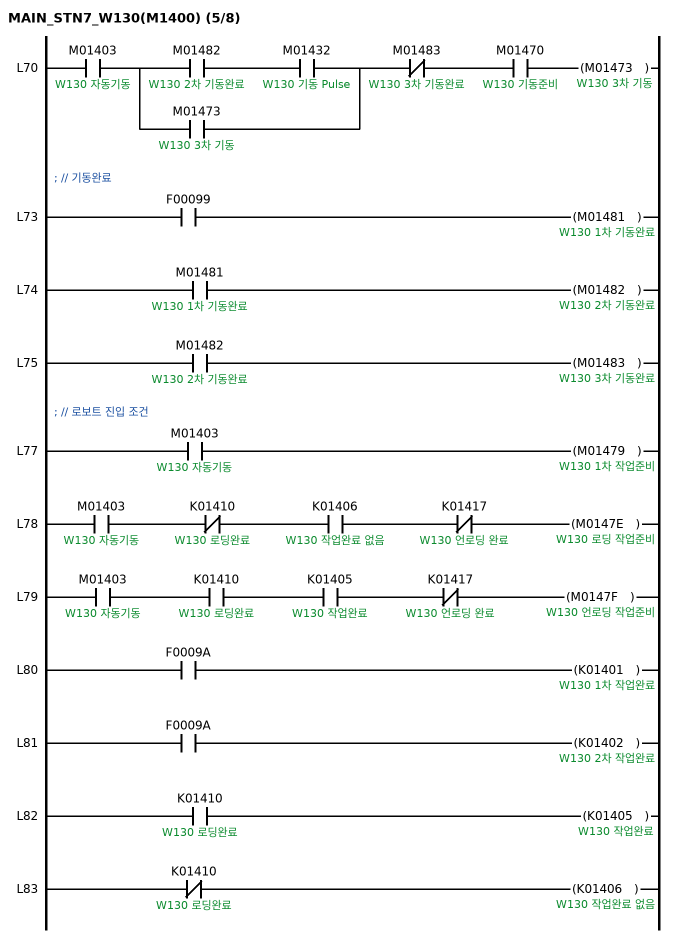
[picture p144: MAIN_STN7_W130(M1400) rungs L70-L83]
; L70
LOAD      M01403	// W130 자동기동
LOAD      M01482	// W130 2차 기동완료
AND       M01432	// W130 기동 Pulse
OR        M01473	// W130 3차 기동
AND LOAD
AND NOT   M01483	// W130 3차 기동완료
AND       M01470	// W130 기동준비
OUT       M01473	// W130 3차 기동
//   // 기동완료
; L73
LOAD      F00099
OUT       M01481	// W130 1차 기동완료
; L74
LOAD      M01481	// W130 1차 기동완료
OUT       M01482	// W130 2차 기동완료
; L75
LOAD      M01482	// W130 2차 기동완료
OUT       M01483	// W130 3차 기동완료
//   // 로보트 진입 조건
; L77
LOAD      M01403	// W130 자동기동
OUT       M01479	// W130 1차 작업준비
; L78
LOAD      M01403	// W130 자동기동
AND NOT   K01410	// W130 로딩완료
AND       K01406	// W130 작업완료 없음
AND NOT   K01417	// W130 언로딩 완료
OUT       M0147E	// W130 로딩 작업준비
; L79
LOAD      M01403	// W130 자동기동
AND       K01410	// W130 로딩완료
AND       K01405	// W130 작업완료
AND NOT   K01417	// W130 언로딩 완료
OUT       M0147F	// W130 언로딩 작업준비
; L80
LOAD      F0009A
OUT       K01401	// W130 1차 작업완료
; L81
LOAD      F0009A
OUT       K01402	// W130 2차 작업완료
; L82
LOAD      K01410	// W130 로딩완료
OUT       K01405	// W130 작업완료
; L83
LOAD NOT  K01410	// W130 로딩완료
OUT       K01406	// W130 작업완료 없음

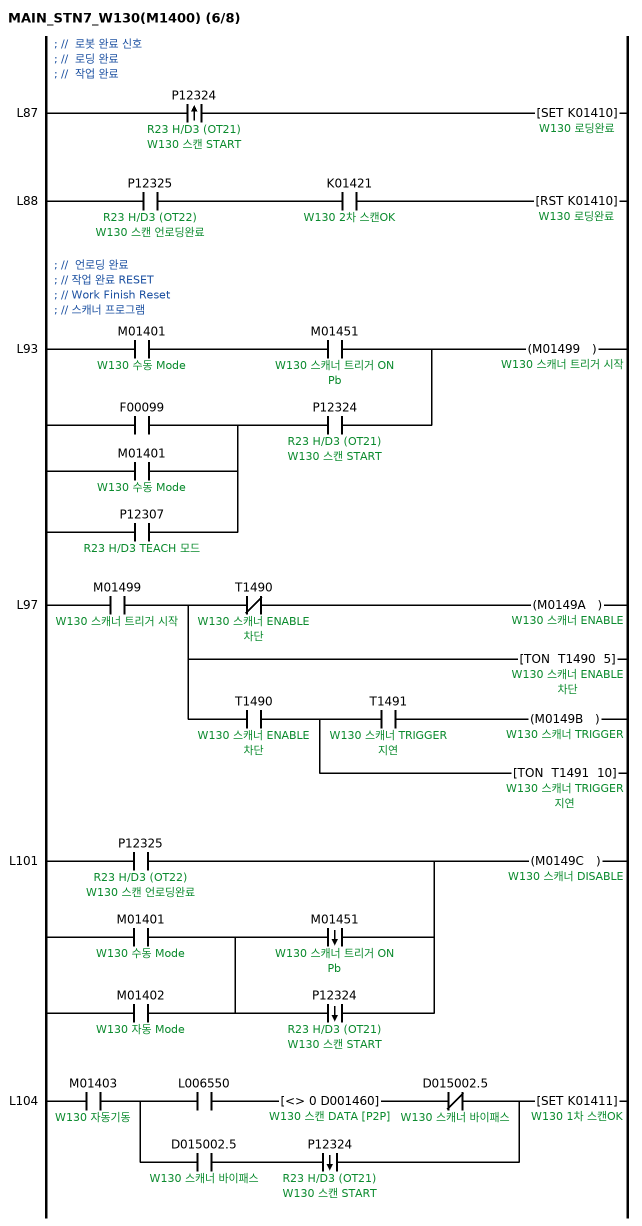
//   //  로봇 완료 신호
//   //  로딩 완료
//   //  작업 완료
; L87
LOADP     P12324	// R23 H/D3 (OT21) W130 스캔 START
SET       K01410	// W130 로딩완료
; L88
LOAD      P12325	// R23 H/D3 (OT22) W130 스캔 언로딩완료
AND       K01421	// W130 2차 스캔OK
RST       K01410	// W130 로딩완료
//   //  언로딩 완료
//     // 작업 완료 RESET
//   // Work Finish Reset
//   // 스캐너 프로그램
; L93
LOAD      M01401	// W130 수동 Mode
AND       M01451	// W130 스캐너 트리거 ON Pb
LOAD      F00099
OR        M01401	// W130 수동 Mode
OR        P12307	// R23 H/D3 TEACH 모드
AND       P12324	// R23 H/D3 (OT21) W130 스캔 START
OR LOAD
OUT       M01499	// W130 스캐너 트리거 시작
; L97
LOAD      M01499	// W130 스캐너 트리거 시작
MPUSH
AND NOT   T1490	// W130 스캐너 ENABLE 차단
OUT       M0149A	// W130 스캐너 ENABLE
MPOP
TON       T1490 5	// W130 스캐너 ENABLE 차단
AND       T1490	// W130 스캐너 ENABLE 차단
MPUSH
AND       T1491	// W130 스캐너 TRIGGER 지연
OUT       M0149B	// W130 스캐너 TRIGGER
MPOP
TON       T1491 10	// W130 스캐너 TRIGGER 지연
; L101
LOAD      P12325	// R23 H/D3 (OT22) W130 스캔 언로딩완료
LOAD      M01401	// W130 수동 Mode
OR        M01402	// W130 자동 Mode
LOADN     M01451	// W130 스캐너 트리거 ON Pb
ORN       P12324	// R23 H/D3 (OT21) W130 스캔 START
AND LOAD
OR LOAD
OUT       M0149C	// W130 스캐너 DISABLE
; L104
LOAD      M01403	// W130 자동기동
LOAD      L006550
AND<>     0 D001460	// W130 스캔 DATA [P2P]
AND NOT   D015002.5	// W130 스캐너 바이패스
LOAD      D015002.5	// W130 스캐너 바이패스
ANDN      P12324	// R23 H/D3 (OT21) W130 스캔 START
OR LOAD
AND LOAD
SET       K01411	// W130 1차 스캔OK

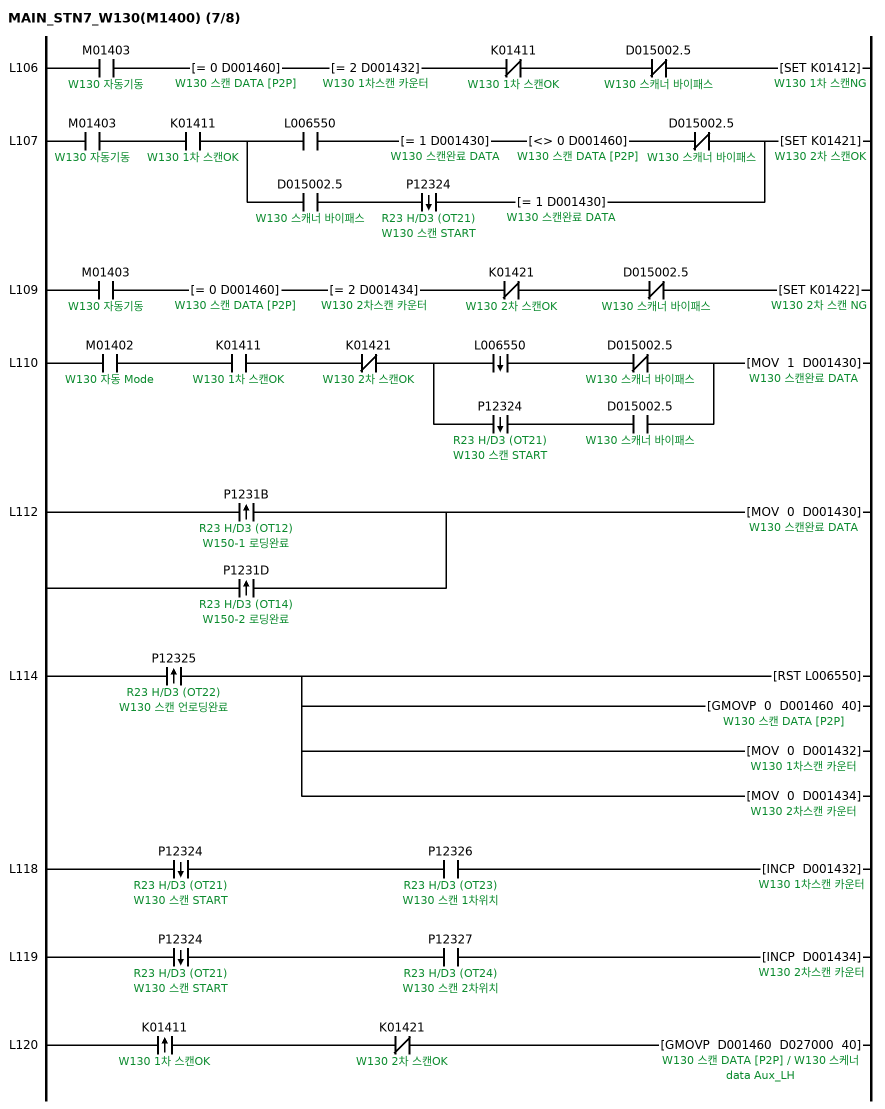
; L106
LOAD      M01403	// W130 자동기동
AND=      0 D001460	// W130 스캔 DATA [P2P]
AND=      2 D001432	// W130 1차스캔 카운터
AND NOT   K01411	// W130 1차 스캔OK
AND NOT   D015002.5	// W130 스캐너 바이패스
SET       K01412	// W130 1차 스캔NG
; L107
LOAD      M01403	// W130 자동기동
AND       K01411	// W130 1차 스캔OK
LOAD      L006550
AND=      1 D001430	// W130 스캔완료 DATA
AND<>     0 D001460	// W130 스캔 DATA [P2P]
AND NOT   D015002.5	// W130 스캐너 바이패스
LOAD      D015002.5	// W130 스캐너 바이패스
ANDN      P12324	// R23 H/D3 (OT21) W130 스캔 START
AND=      1 D001430	// W130 스캔완료 DATA
OR LOAD
AND LOAD
SET       K01421	// W130 2차 스캔OK
; L109
LOAD      M01403	// W130 자동기동
AND=      0 D001460	// W130 스캔 DATA [P2P]
AND=      2 D001434	// W130 2차스캔 카운터
AND NOT   K01421	// W130 2차 스캔OK
AND NOT   D015002.5	// W130 스캐너 바이패스
SET       K01422	// W130 2차 스캔 NG
; L110
LOAD      M01402	// W130 자동 Mode
AND       K01411	// W130 1차 스캔OK
AND NOT   K01421	// W130 2차 스캔OK
LOADN     L006550
AND NOT   D015002.5	// W130 스캐너 바이패스
LOADN     P12324	// R23 H/D3 (OT21) W130 스캔 START
AND       D015002.5	// W130 스캐너 바이패스
OR LOAD
AND LOAD
MOV       1 D001430	// W130 스캔완료 DATA
; L112
LOADP     P1231B	// R23 H/D3 (OT12) W150-1 로딩완료
ORP       P1231D	// R23 H/D3 (OT14) W150-2 로딩완료
MOV       0 D001430	// W130 스캔완료 DATA
; L114
LOADP     P12325	// R23 H/D3 (OT22) W130 스캔 언로딩완료
RST       L006550
GMOVP     0 D001460 40	// W130 스캔 DATA [P2P]
MOV       0 D001432	// W130 1차스캔 카운터
MOV       0 D001434	// W130 2차스캔 카운터
; L118
LOADN     P12324	// R23 H/D3 (OT21) W130 스캔 START
AND       P12326	// R23 H/D3 (OT23) W130 스캔 1차위치
INCP      D001432	// W130 1차스캔 카운터
; L119
LOADN     P12324	// R23 H/D3 (OT21) W130 스캔 START
AND       P12327	// R23 H/D3 (OT24) W130 스캔 2차위치
INCP      D001434	// W130 2차스캔 카운터
; L120
LOADP     K01411	// W130 1차 스캔OK
AND NOT   K01421	// W130 2차 스캔OK
GMOVP     D001460 D027000 40	// W130 스캔 DATA [P2P] / W130 스케너 data Aux_LH

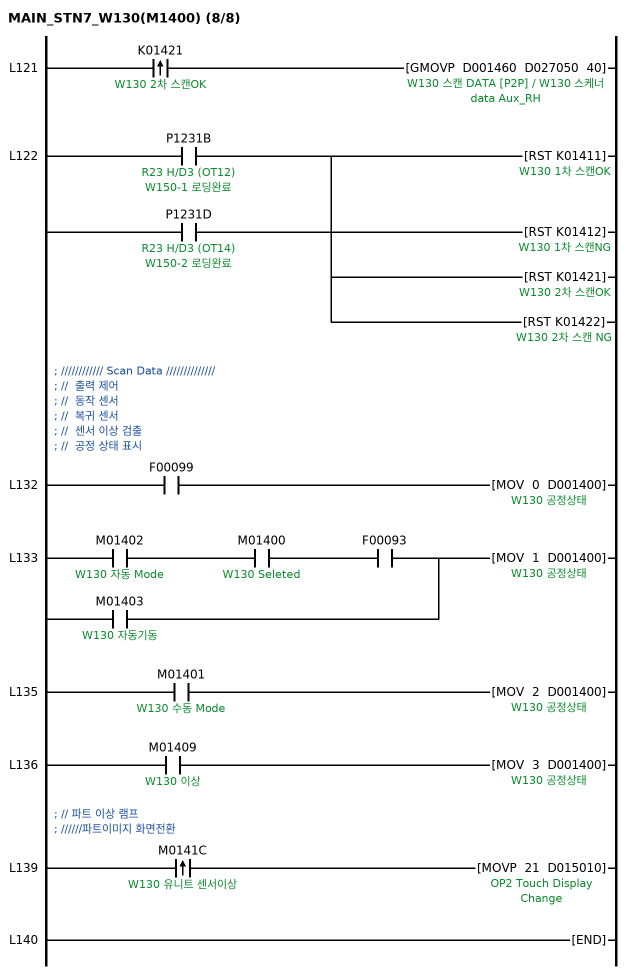
; L121
LOADP     K01421	// W130 2차 스캔OK
GMOVP     D001460 D027050 40	// W130 스캔 DATA [P2P] / W130 스케너 data Aux_RH
; L122
LOAD      P1231B	// R23 H/D3 (OT12) W150-1 로딩완료
OR        P1231D	// R23 H/D3 (OT14) W150-2 로딩완료
RST       K01411	// W130 1차 스캔OK
RST       K01412	// W130 1차 스캔NG
RST       K01421	// W130 2차 스캔OK
RST       K01422	// W130 2차 스캔 NG
// //////////// Scan Data //////////////
//     //  출력 제어
//   //  동작 센서
//   //  복귀 센서
//     //  센서 이상 검출
//   //  공정 상태 표시
; L132
LOAD      F00099
MOV       0 D001400	// W130 공정상태
; L133
LOAD      M01402	// W130 자동 Mode
AND       M01400	// W130 Seleted
AND       F00093
OR        M01403	// W130 자동기동
MOV       1 D001400	// W130 공정상태
; L135
LOAD      M01401	// W130 수동 Mode
MOV       2 D001400	// W130 공정상태
; L136
LOAD      M01409	// W130 이상
MOV       3 D001400	// W130 공정상태
//   // 파트 이상 램프
// //////파트이미지 화면전환
; L139
LOADP     M0141C	// W130 유니트 센서이상
MOVP      21 D015010	// OP2 Touch Display Change
; L140
END

PROGRAM MAIN_STN8_W150-1(M800) (task: 스캔 프로그램)

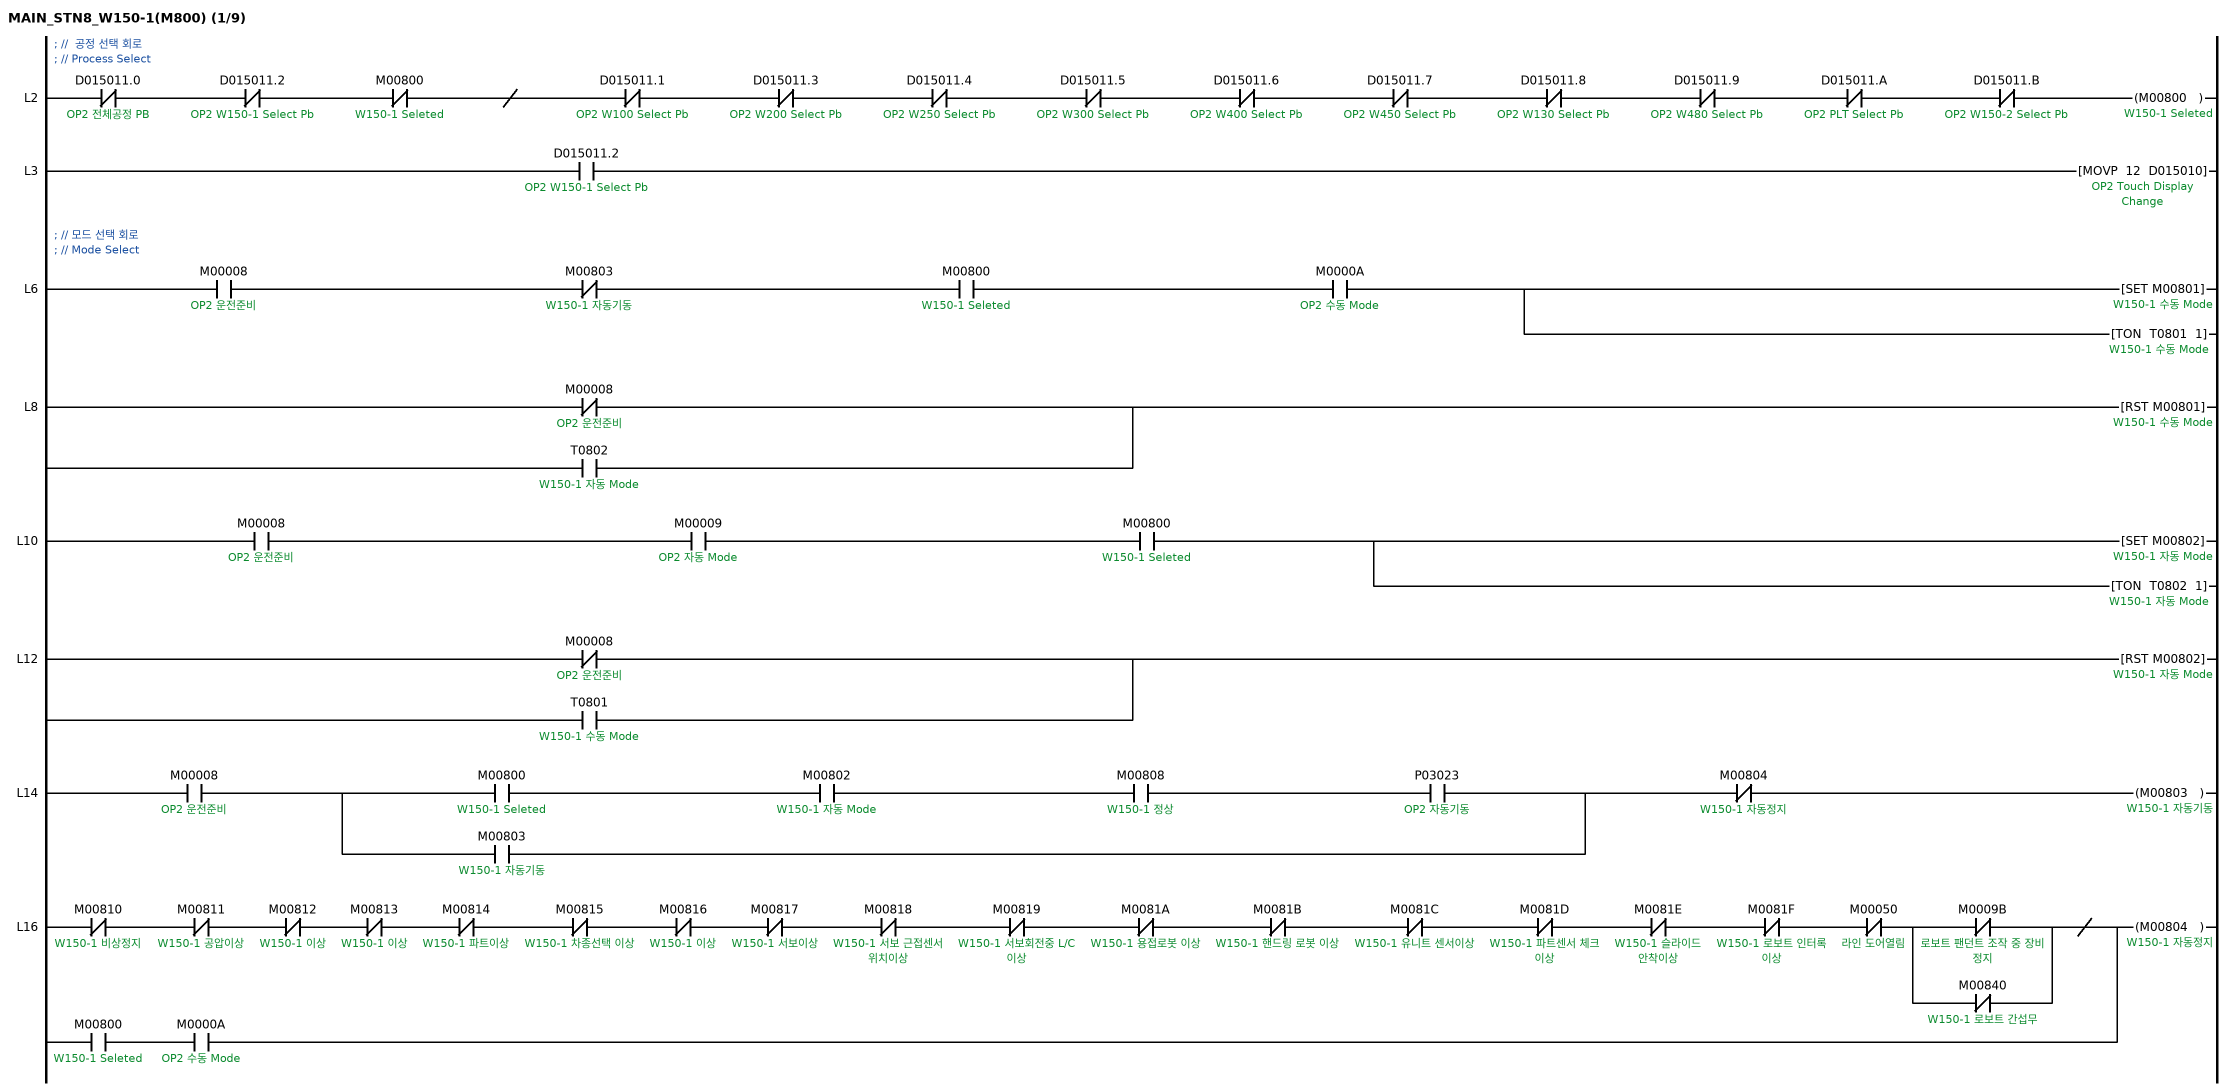
//   //  공정 선택 회로
//   // Process Select
; L2
LOAD NOT  D015011.0	// OP2 전체공정 PB
AND NOT   D015011.2	// OP2 W150-1 Select Pb
AND NOT   M00800	// W150-1 Seleted
NOT
AND NOT   D015011.1	// OP2 W100 Select Pb
AND NOT   D015011.3	// OP2 W200 Select Pb
AND NOT   D015011.4	// OP2 W250 Select Pb
AND NOT   D015011.5	// OP2 W300 Select Pb
AND NOT   D015011.6	// OP2 W400 Select Pb
AND NOT   D015011.7	// OP2 W450 Select Pb
AND NOT   D015011.8	// OP2 W130 Select Pb
AND NOT   D015011.9	// OP2 W480 Select Pb
AND NOT   D015011.A	// OP2 PLT Select Pb
AND NOT   D015011.B	// OP2 W150-2 Select Pb
OUT       M00800	// W150-1 Seleted
; L3
LOAD      D015011.2	// OP2 W150-1 Select Pb
MOVP      12 D015010	// OP2 Touch Display Change
// // 모드 선택 회로
//   // Mode Select
; L6
LOAD      M00008	// OP2 운전준비
AND NOT   M00803	// W150-1 자동기동
AND       M00800	// W150-1 Seleted
AND       M0000A	// OP2 수동 Mode
SET       M00801	// W150-1 수동 Mode
TON       T0801 1	// W150-1 수동 Mode
; L8
LOAD NOT  M00008	// OP2 운전준비
OR        T0802	// W150-1 자동 Mode
RST       M00801	// W150-1 수동 Mode
; L10
LOAD      M00008	// OP2 운전준비
AND       M00009	// OP2 자동 Mode
AND       M00800	// W150-1 Seleted
SET       M00802	// W150-1 자동 Mode
TON       T0802 1	// W150-1 자동 Mode
; L12
LOAD NOT  M00008	// OP2 운전준비
OR        T0801	// W150-1 수동 Mode
RST       M00802	// W150-1 자동 Mode
; L14
LOAD      M00008	// OP2 운전준비
LOAD      M00800	// W150-1 Seleted
AND       M00802	// W150-1 자동 Mode
AND       M00808	// W150-1 정상
AND       P03023	// OP2 자동기동
OR        M00803	// W150-1 자동기동
AND LOAD
AND NOT   M00804	// W150-1 자동정지
OUT       M00803	// W150-1 자동기동
; L16
LOAD NOT  M00810	// W150-1 비상정지
AND NOT   M00811	// W150-1 공압이상
AND NOT   M00812	// W150-1 이상
AND NOT   M00813	// W150-1 이상
AND NOT   M00814	// W150-1 파트이상
AND NOT   M00815	// W150-1 차종선택 이상
AND NOT   M00816	// W150-1 이상
AND NOT   M00817	// W150-1 서보이상
AND NOT   M00818	// W150-1 서보 근접센서 위치이상
AND NOT   M00819	// W150-1 서보회전중 L/C 이상
AND NOT   M0081A	// W150-1 용접로봇 이상
AND NOT   M0081B	// W150-1 핸드링 로봇 이상
AND NOT   M0081C	// W150-1 유니트 센서이상
AND NOT   M0081D	// W150-1 파트센서 체크 이상
AND NOT   M0081E	// W150-1 슬라이드 안착이상
AND NOT   M0081F	// W150-1 로보트 인터록 이상
AND NOT   M00050	// 라인 도어열림
LOAD NOT  M0009B	// 로보트 팬던트 조작 중 장비 정지
OR NOT    M00840	// W150-1 로보트 간섭무
AND LOAD
NOT
LOAD      M00800	// W150-1 Seleted
AND       M0000A	// OP2 수동 Mode
OR LOAD
OUT       M00804	// W150-1 자동정지

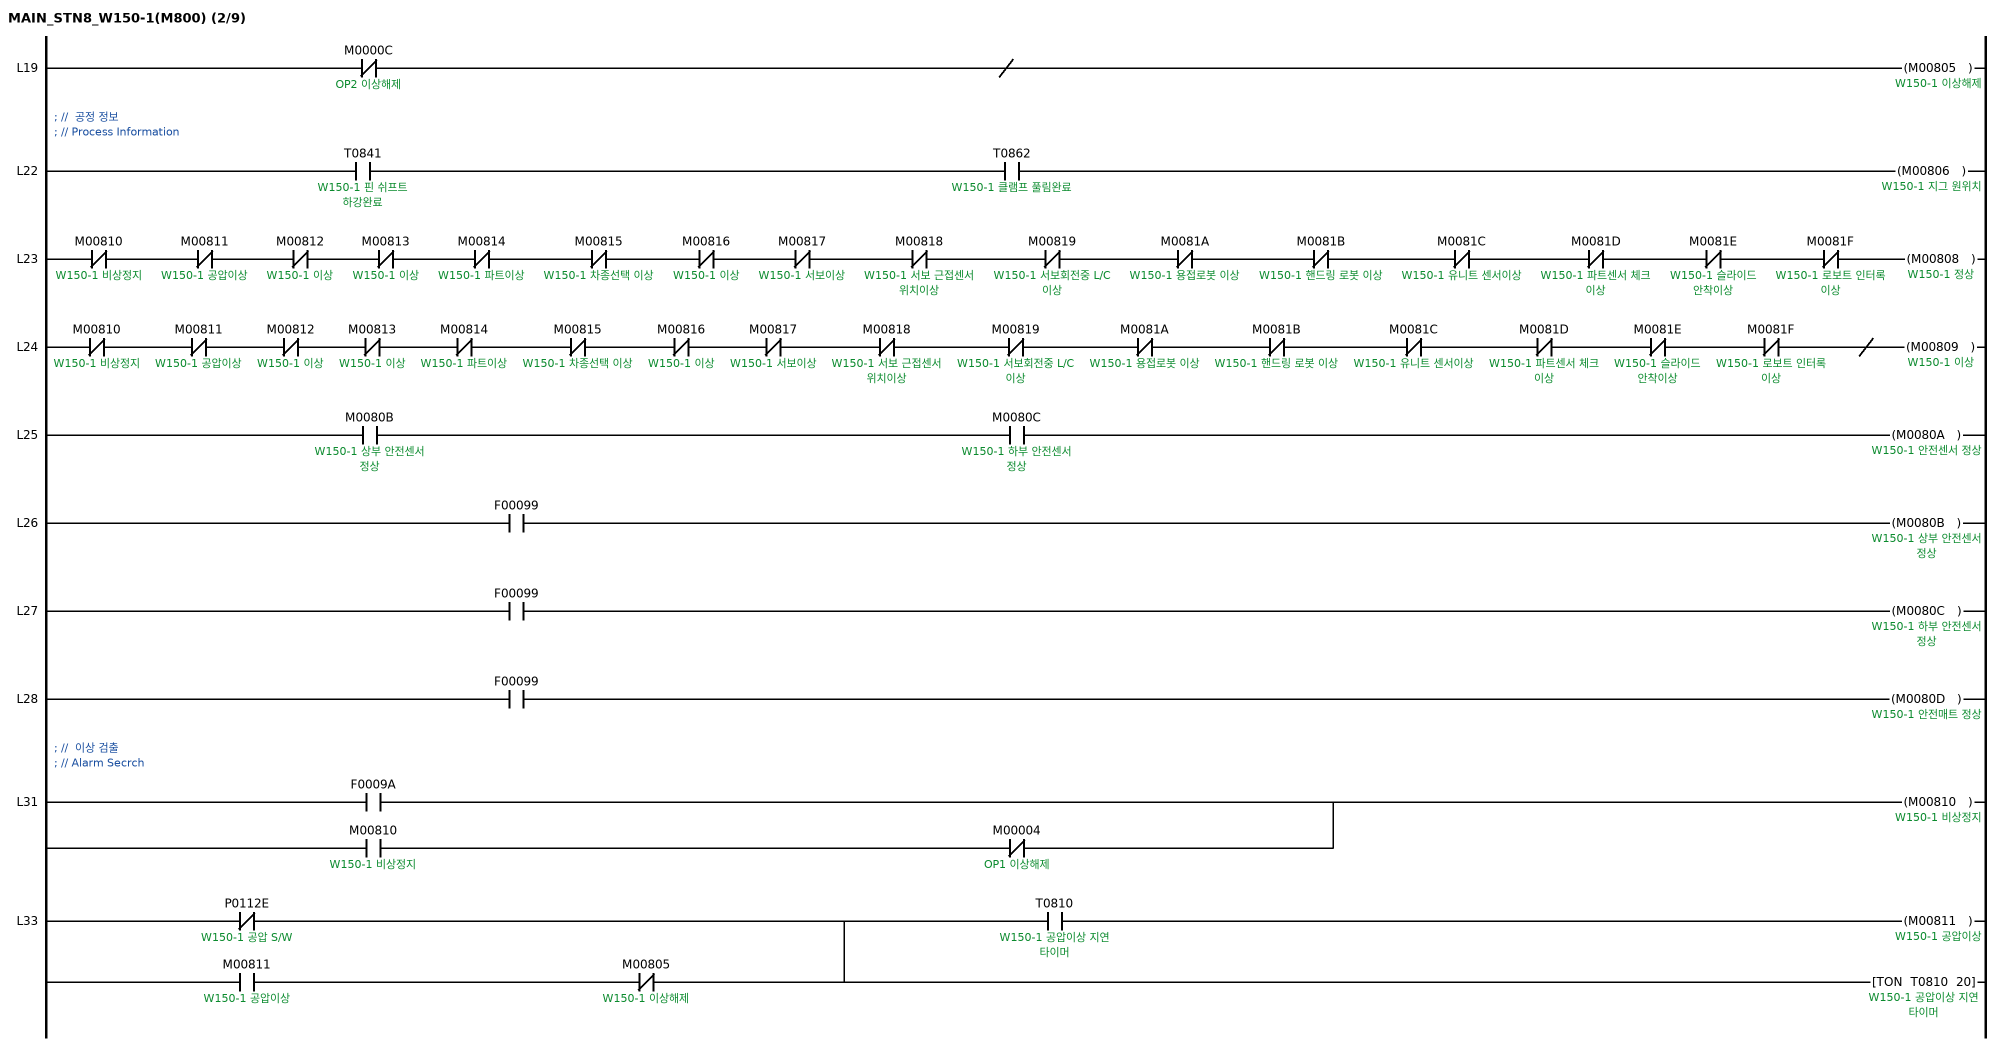
; L19
LOAD NOT  M0000C	// OP2 이상해제
NOT
OUT       M00805	// W150-1 이상해제
//   //  공정 정보
//   // Process Information
; L22
LOAD      T0841	// W150-1 핀 쉬프트 하강완료
AND       T0862	// W150-1 클램프 풀림완료
OUT       M00806	// W150-1 지그 원위치
; L23
LOAD NOT  M00810	// W150-1 비상정지
AND NOT   M00811	// W150-1 공압이상
AND NOT   M00812	// W150-1 이상
AND NOT   M00813	// W150-1 이상
AND NOT   M00814	// W150-1 파트이상
AND NOT   M00815	// W150-1 차종선택 이상
AND NOT   M00816	// W150-1 이상
AND NOT   M00817	// W150-1 서보이상
AND NOT   M00818	// W150-1 서보 근접센서 위치이상
AND NOT   M00819	// W150-1 서보회전중 L/C 이상
AND NOT   M0081A	// W150-1 용접로봇 이상
AND NOT   M0081B	// W150-1 핸드링 로봇 이상
AND NOT   M0081C	// W150-1 유니트 센서이상
AND NOT   M0081D	// W150-1 파트센서 체크 이상
AND NOT   M0081E	// W150-1 슬라이드 안착이상
AND NOT   M0081F	// W150-1 로보트 인터록 이상
OUT       M00808	// W150-1 정상
; L24
LOAD NOT  M00810	// W150-1 비상정지
AND NOT   M00811	// W150-1 공압이상
AND NOT   M00812	// W150-1 이상
AND NOT   M00813	// W150-1 이상
AND NOT   M00814	// W150-1 파트이상
AND NOT   M00815	// W150-1 차종선택 이상
AND NOT   M00816	// W150-1 이상
AND NOT   M00817	// W150-1 서보이상
AND NOT   M00818	// W150-1 서보 근접센서 위치이상
AND NOT   M00819	// W150-1 서보회전중 L/C 이상
AND NOT   M0081A	// W150-1 용접로봇 이상
AND NOT   M0081B	// W150-1 핸드링 로봇 이상
AND NOT   M0081C	// W150-1 유니트 센서이상
AND NOT   M0081D	// W150-1 파트센서 체크 이상
AND NOT   M0081E	// W150-1 슬라이드 안착이상
AND NOT   M0081F	// W150-1 로보트 인터록 이상
NOT
OUT       M00809	// W150-1 이상
; L25
LOAD      M0080B	// W150-1 상부 안전센서 정상
AND       M0080C	// W150-1 하부 안전센서 정상
OUT       M0080A	// W150-1 안전센서 정상
; L26
LOAD      F00099
OUT       M0080B	// W150-1 상부 안전센서 정상
; L27
LOAD      F00099
OUT       M0080C	// W150-1 하부 안전센서 정상
; L28
LOAD      F00099
OUT       M0080D	// W150-1 안전매트 정상
//   //  이상 검출
//   // Alarm Secrch
; L31
LOAD      F0009A
LOAD      M00810	// W150-1 비상정지
AND NOT   M00004	// OP1 이상해제
OR LOAD
OUT       M00810	// W150-1 비상정지
; L33
LOAD NOT  P0112E	// W150-1 공압 S/W
LOAD      M00811	// W150-1 공압이상
AND NOT   M00805	// W150-1 이상해제
OR LOAD
MPUSH
AND       T0810	// W150-1 공압이상 지연 타이머
OUT       M00811	// W150-1 공압이상
MPOP
TON       T0810 20	// W150-1 공압이상 지연 타이머

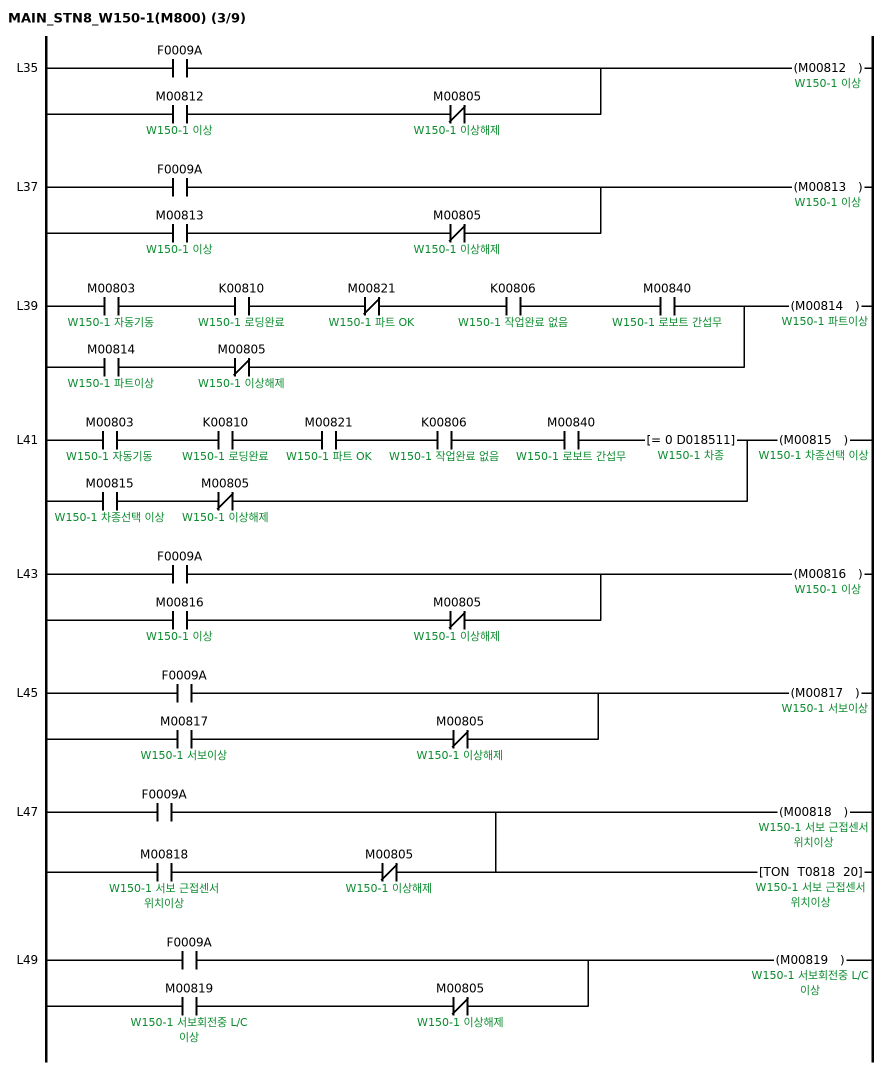
; L35
LOAD      F0009A
LOAD      M00812	// W150-1 이상
AND NOT   M00805	// W150-1 이상해제
OR LOAD
OUT       M00812	// W150-1 이상
; L37
LOAD      F0009A
LOAD      M00813	// W150-1 이상
AND NOT   M00805	// W150-1 이상해제
OR LOAD
OUT       M00813	// W150-1 이상
; L39
LOAD      M00803	// W150-1 자동기동
AND       K00810	// W150-1 로딩완료
AND NOT   M00821	// W150-1 파트 OK
AND       K00806	// W150-1 작업완료 없음
AND       M00840	// W150-1 로보트 간섭무
LOAD      M00814	// W150-1 파트이상
AND NOT   M00805	// W150-1 이상해제
OR LOAD
OUT       M00814	// W150-1 파트이상
; L41
LOAD      M00803	// W150-1 자동기동
AND       K00810	// W150-1 로딩완료
AND       M00821	// W150-1 파트 OK
AND       K00806	// W150-1 작업완료 없음
AND       M00840	// W150-1 로보트 간섭무
AND=      0 D018511	// W150-1 차종
LOAD      M00815	// W150-1 차종선택 이상
AND NOT   M00805	// W150-1 이상해제
OR LOAD
OUT       M00815	// W150-1 차종선택 이상
; L43
LOAD      F0009A
LOAD      M00816	// W150-1 이상
AND NOT   M00805	// W150-1 이상해제
OR LOAD
OUT       M00816	// W150-1 이상
; L45
LOAD      F0009A
LOAD      M00817	// W150-1 서보이상
AND NOT   M00805	// W150-1 이상해제
OR LOAD
OUT       M00817	// W150-1 서보이상
; L47
LOAD      F0009A
LOAD      M00818	// W150-1 서보 근접센서 위치이상
AND NOT   M00805	// W150-1 이상해제
OR LOAD
OUT       M00818	// W150-1 서보 근접센서 위치이상
TON       T0818 20	// W150-1 서보 근접센서 위치이상
; L49
LOAD      F0009A
LOAD      M00819	// W150-1 서보회전중 L/C 이상
AND NOT   M00805	// W150-1 이상해제
OR LOAD
OUT       M00819	// W150-1 서보회전중 L/C 이상

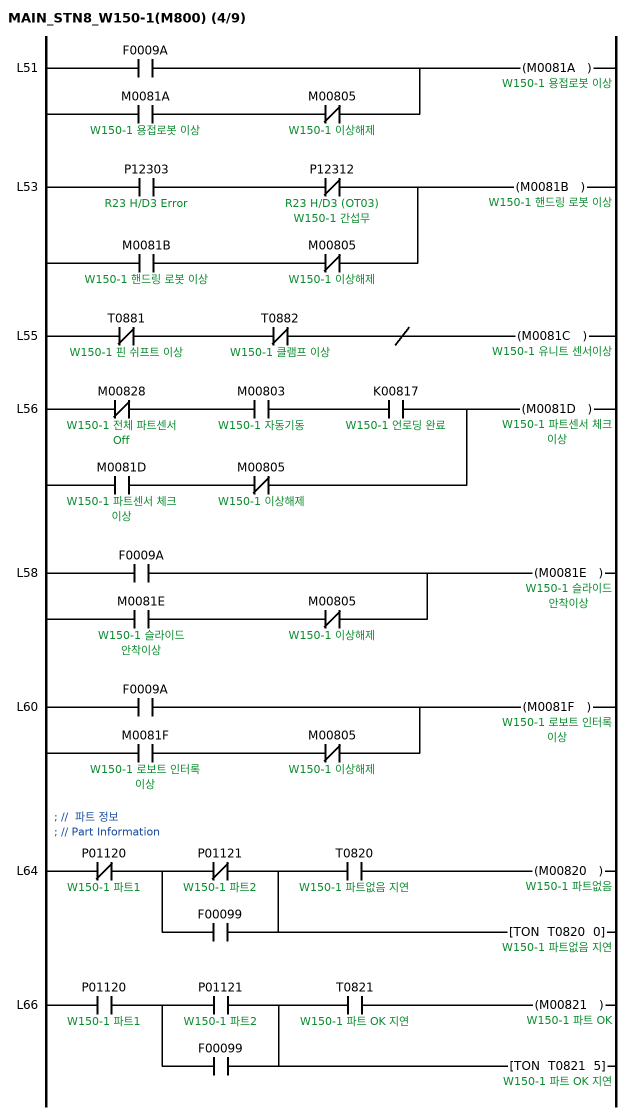
; L51
LOAD      F0009A
LOAD      M0081A	// W150-1 용접로봇 이상
AND NOT   M00805	// W150-1 이상해제
OR LOAD
OUT       M0081A	// W150-1 용접로봇 이상
; L53
LOAD      P12303	// R23 H/D3 Error
AND NOT   P12312	// R23 H/D3 (OT03) W150-1 간섭무
LOAD      M0081B	// W150-1 핸드링 로봇 이상
AND NOT   M00805	// W150-1 이상해제
OR LOAD
OUT       M0081B	// W150-1 핸드링 로봇 이상
; L55
LOAD NOT  T0881	// W150-1 핀 쉬프트 이상
AND NOT   T0882	// W150-1 클램프 이상
NOT
OUT       M0081C	// W150-1 유니트 센서이상
; L56
LOAD NOT  M00828	// W150-1 전체 파트센서 Off
AND       M00803	// W150-1 자동기동
AND       K00817	// W150-1 언로딩 완료
LOAD      M0081D	// W150-1 파트센서 체크 이상
AND NOT   M00805	// W150-1 이상해제
OR LOAD
OUT       M0081D	// W150-1 파트센서 체크 이상
; L58
LOAD      F0009A
LOAD      M0081E	// W150-1 슬라이드 안착이상
AND NOT   M00805	// W150-1 이상해제
OR LOAD
OUT       M0081E	// W150-1 슬라이드 안착이상
; L60
LOAD      F0009A
LOAD      M0081F	// W150-1 로보트 인터록 이상
AND NOT   M00805	// W150-1 이상해제
OR LOAD
OUT       M0081F	// W150-1 로보트 인터록 이상
//   //  파트 정보
//   // Part Information
; L64
LOAD NOT  P01120	// W150-1 파트1
LOAD NOT  P01121	// W150-1 파트2
OR        F00099
AND LOAD
MPUSH
AND       T0820	// W150-1 파트없음 지연
OUT       M00820	// W150-1 파트없음
MPOP
TON       T0820 0	// W150-1 파트없음 지연
; L66
LOAD      P01120	// W150-1 파트1
LOAD      P01121	// W150-1 파트2
OR        F00099
AND LOAD
MPUSH
AND       T0821	// W150-1 파트 OK 지연
OUT       M00821	// W150-1 파트 OK
MPOP
TON       T0821 5	// W150-1 파트 OK 지연

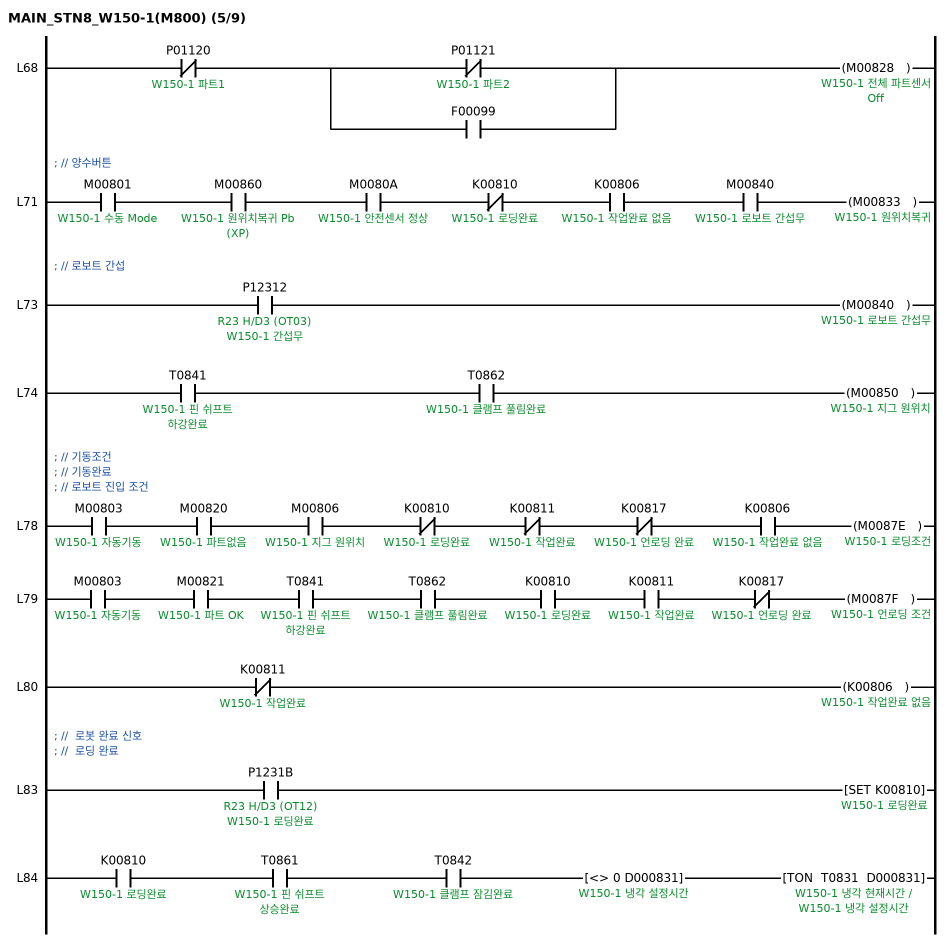
; L68
LOAD NOT  P01120	// W150-1 파트1
LOAD NOT  P01121	// W150-1 파트2
OR        F00099
AND LOAD
OUT       M00828	// W150-1 전체 파트센서 Off
//   // 양수버튼
; L71
LOAD      M00801	// W150-1 수동 Mode
AND       M00860	// W150-1 원위치복귀 Pb (XP)
AND       M0080A	// W150-1 안전센서 정상
AND NOT   K00810	// W150-1 로딩완료
AND       K00806	// W150-1 작업완료 없음
AND       M00840	// W150-1 로보트 간섭무
OUT       M00833	// W150-1 원위치복귀
//   // 로보트 간섭
; L73
LOAD      P12312	// R23 H/D3 (OT03) W150-1 간섭무
OUT       M00840	// W150-1 로보트 간섭무
; L74
LOAD      T0841	// W150-1 핀 쉬프트 하강완료
AND       T0862	// W150-1 클램프 풀림완료
OUT       M00850	// W150-1 지그 원위치
//   // 기동조건
//   // 기동완료
//   // 로보트 진입 조건
; L78
LOAD      M00803	// W150-1 자동기동
AND       M00820	// W150-1 파트없음
AND       M00806	// W150-1 지그 원위치
AND NOT   K00810	// W150-1 로딩완료
AND NOT   K00811	// W150-1 작업완료
AND NOT   K00817	// W150-1 언로딩 완료
AND       K00806	// W150-1 작업완료 없음
OUT       M0087E	// W150-1 로딩조건
; L79
LOAD      M00803	// W150-1 자동기동
AND       M00821	// W150-1 파트 OK
AND       T0841	// W150-1 핀 쉬프트 하강완료
AND       T0862	// W150-1 클램프 풀림완료
AND       K00810	// W150-1 로딩완료
AND       K00811	// W150-1 작업완료
AND NOT   K00817	// W150-1 언로딩 완료
OUT       M0087F	// W150-1 언로딩 조건
; L80
LOAD NOT  K00811	// W150-1 작업완료
OUT       K00806	// W150-1 작업완료 없음
//   //  로봇 완료 신호
//   //  로딩 완료
; L83
LOAD      P1231B	// R23 H/D3 (OT12) W150-1 로딩완료
SET       K00810	// W150-1 로딩완료
; L84
LOAD      K00810	// W150-1 로딩완료
AND       T0861	// W150-1 핀 쉬프트 상승완료
AND       T0842	// W150-1 클램프 잠김완료
AND<>     0 D000831	// W150-1 냉각 설정시간
TON       T0831 D000831	// W150-1 냉각 현재시간 / W150-1 냉각 설정시간

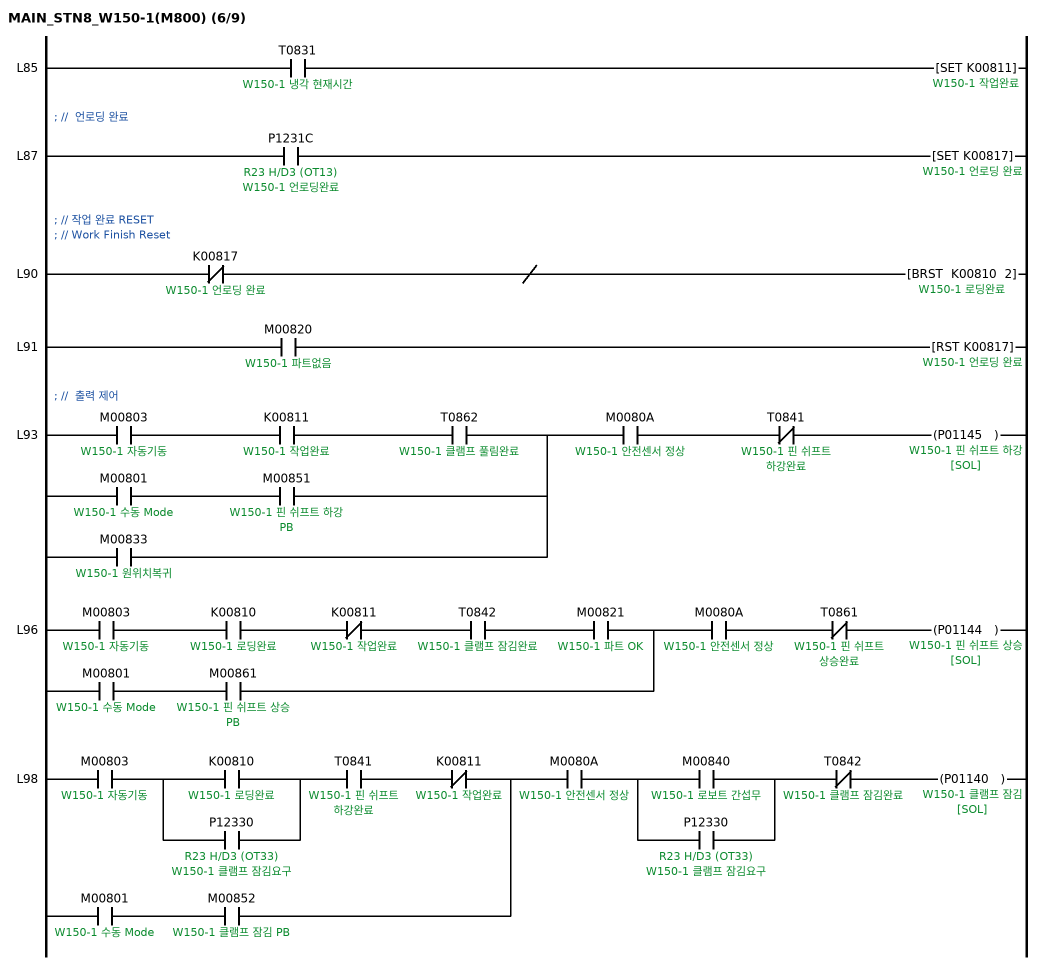
; L85
LOAD      T0831	// W150-1 냉각 현재시간
SET       K00811	// W150-1 작업완료
//   //  언로딩 완료
; L87
LOAD      P1231C	// R23 H/D3 (OT13) W150-1 언로딩완료
SET       K00817	// W150-1 언로딩 완료
//     // 작업 완료 RESET
//   // Work Finish Reset
; L90
LOAD NOT  K00817	// W150-1 언로딩 완료
NOT
BRST      K00810 2	// W150-1 로딩완료
; L91
LOAD      M00820	// W150-1 파트없음
RST       K00817	// W150-1 언로딩 완료
//     //  출력 제어
; L93
LOAD      M00803	// W150-1 자동기동
AND       K00811	// W150-1 작업완료
AND       T0862	// W150-1 클램프 풀림완료
LOAD      M00801	// W150-1 수동 Mode
AND       M00851	// W150-1 핀 쉬프트 하강 PB
OR LOAD
OR        M00833	// W150-1 원위치복귀
AND       M0080A	// W150-1 안전센서 정상
AND NOT   T0841	// W150-1 핀 쉬프트 하강완료
OUT       P01145	// W150-1 핀 쉬프트 하강 [SOL]
; L96
LOAD      M00803	// W150-1 자동기동
AND       K00810	// W150-1 로딩완료
AND NOT   K00811	// W150-1 작업완료
AND       T0842	// W150-1 클램프 잠김완료
AND       M00821	// W150-1 파트 OK
LOAD      M00801	// W150-1 수동 Mode
AND       M00861	// W150-1 핀 쉬프트 상승 PB
OR LOAD
AND       M0080A	// W150-1 안전센서 정상
AND NOT   T0861	// W150-1 핀 쉬프트 상승완료
OUT       P01144	// W150-1 핀 쉬프트 상승 [SOL]
; L98
LOAD      M00803	// W150-1 자동기동
LOAD      K00810	// W150-1 로딩완료
OR        P12330	// R23 H/D3 (OT33) W150-1 클램프 잠김요구
AND LOAD
AND       T0841	// W150-1 핀 쉬프트 하강완료
AND NOT   K00811	// W150-1 작업완료
LOAD      M00801	// W150-1 수동 Mode
AND       M00852	// W150-1 클램프 잠김 PB
OR LOAD
AND       M0080A	// W150-1 안전센서 정상
LOAD      M00840	// W150-1 로보트 간섭무
OR        P12330	// R23 H/D3 (OT33) W150-1 클램프 잠김요구
AND LOAD
AND NOT   T0842	// W150-1 클램프 잠김완료
OUT       P01140	// W150-1 클램프 잠김 [SOL]

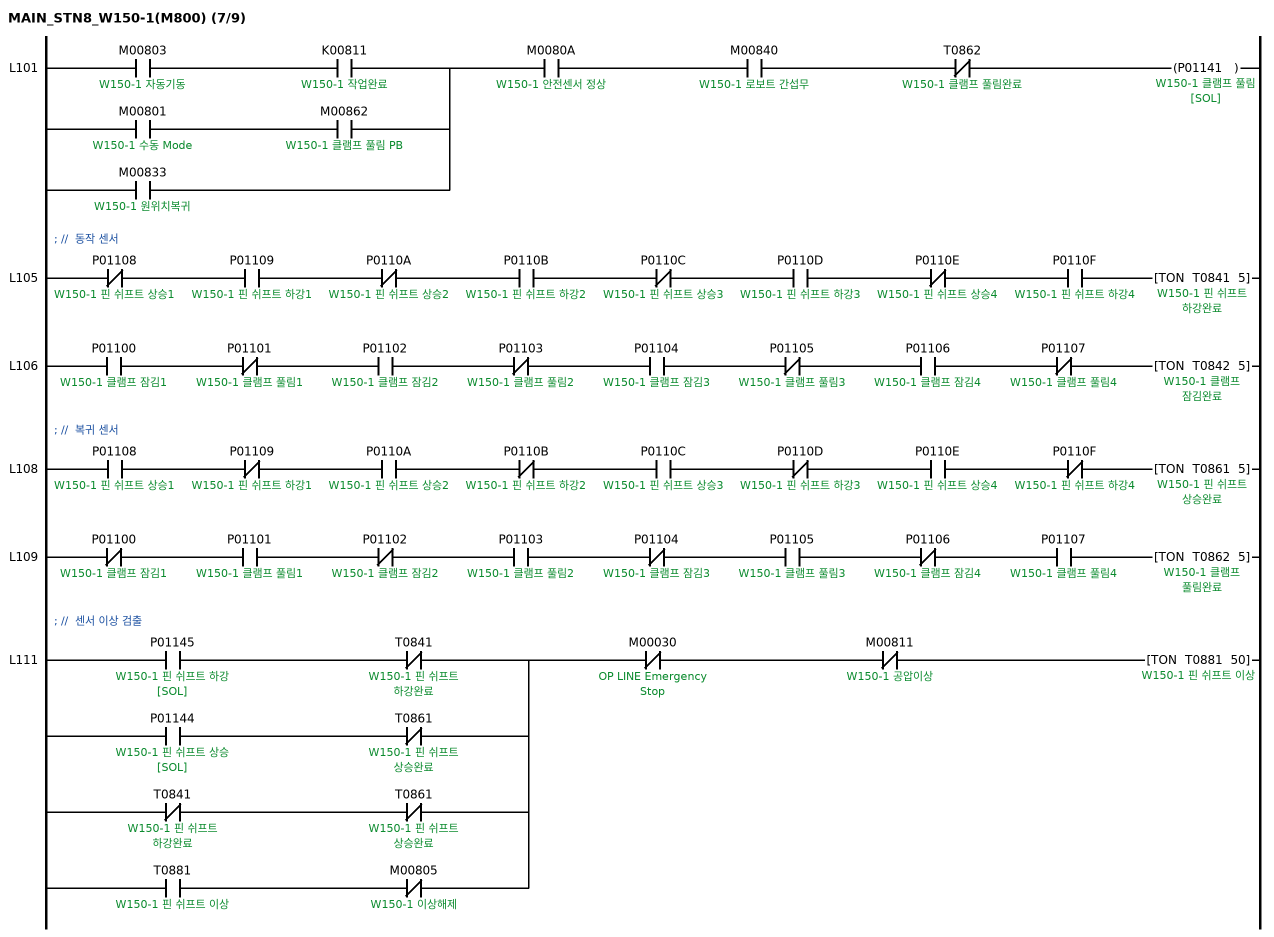
; L101
LOAD      M00803	// W150-1 자동기동
AND       K00811	// W150-1 작업완료
LOAD      M00801	// W150-1 수동 Mode
AND       M00862	// W150-1 클램프 풀림 PB
OR LOAD
OR        M00833	// W150-1 원위치복귀
AND       M0080A	// W150-1 안전센서 정상
AND       M00840	// W150-1 로보트 간섭무
AND NOT   T0862	// W150-1 클램프 풀림완료
OUT       P01141	// W150-1 클램프 풀림 [SOL]
//   //  동작 센서
; L105
LOAD NOT  P01108	// W150-1 핀 쉬프트 상승1
AND       P01109	// W150-1 핀 쉬프트 하강1
AND NOT   P0110A	// W150-1 핀 쉬프트 상승2
AND       P0110B	// W150-1 핀 쉬프트 하강2
AND NOT   P0110C	// W150-1 핀 쉬프트 상승3
AND       P0110D	// W150-1 핀 쉬프트 하강3
AND NOT   P0110E	// W150-1 핀 쉬프트 상승4
AND       P0110F	// W150-1 핀 쉬프트 하강4
TON       T0841 5	// W150-1 핀 쉬프트 하강완료
; L106
LOAD      P01100	// W150-1 클램프 잠김1
AND NOT   P01101	// W150-1 클램프 풀림1
AND       P01102	// W150-1 클램프 잠김2
AND NOT   P01103	// W150-1 클램프 풀림2
AND       P01104	// W150-1 클램프 잠김3
AND NOT   P01105	// W150-1 클램프 풀림3
AND       P01106	// W150-1 클램프 잠김4
AND NOT   P01107	// W150-1 클램프 풀림4
TON       T0842 5	// W150-1 클램프 잠김완료
//   //  복귀 센서
; L108
LOAD      P01108	// W150-1 핀 쉬프트 상승1
AND NOT   P01109	// W150-1 핀 쉬프트 하강1
AND       P0110A	// W150-1 핀 쉬프트 상승2
AND NOT   P0110B	// W150-1 핀 쉬프트 하강2
AND       P0110C	// W150-1 핀 쉬프트 상승3
AND NOT   P0110D	// W150-1 핀 쉬프트 하강3
AND       P0110E	// W150-1 핀 쉬프트 상승4
AND NOT   P0110F	// W150-1 핀 쉬프트 하강4
TON       T0861 5	// W150-1 핀 쉬프트 상승완료
; L109
LOAD NOT  P01100	// W150-1 클램프 잠김1
AND       P01101	// W150-1 클램프 풀림1
AND NOT   P01102	// W150-1 클램프 잠김2
AND       P01103	// W150-1 클램프 풀림2
AND NOT   P01104	// W150-1 클램프 잠김3
AND       P01105	// W150-1 클램프 풀림3
AND NOT   P01106	// W150-1 클램프 잠김4
AND       P01107	// W150-1 클램프 풀림4
TON       T0862 5	// W150-1 클램프 풀림완료
//     //  센서 이상 검출
; L111
LOAD      P01145	// W150-1 핀 쉬프트 하강 [SOL]
AND NOT   T0841	// W150-1 핀 쉬프트 하강완료
LOAD      P01144	// W150-1 핀 쉬프트 상승 [SOL]
AND NOT   T0861	// W150-1 핀 쉬프트 상승완료
OR LOAD
LOAD NOT  T0841	// W150-1 핀 쉬프트 하강완료
AND NOT   T0861	// W150-1 핀 쉬프트 상승완료
OR LOAD
LOAD      T0881	// W150-1 핀 쉬프트 이상
AND NOT   M00805	// W150-1 이상해제
OR LOAD
AND NOT   M00030	// OP LINE Emergency Stop
AND NOT   M00811	// W150-1 공압이상
TON       T0881 50	// W150-1 핀 쉬프트 이상

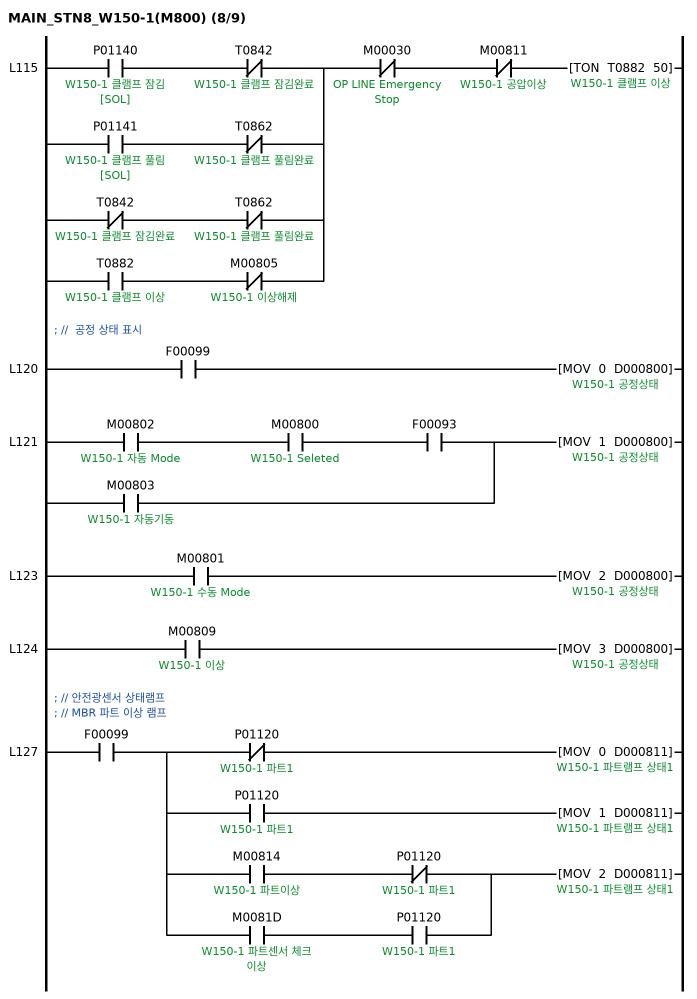
; L115
LOAD      P01140	// W150-1 클램프 잠김 [SOL]
AND NOT   T0842	// W150-1 클램프 잠김완료
LOAD      P01141	// W150-1 클램프 풀림 [SOL]
AND NOT   T0862	// W150-1 클램프 풀림완료
OR LOAD
LOAD NOT  T0842	// W150-1 클램프 잠김완료
AND NOT   T0862	// W150-1 클램프 풀림완료
OR LOAD
LOAD      T0882	// W150-1 클램프 이상
AND NOT   M00805	// W150-1 이상해제
OR LOAD
AND NOT   M00030	// OP LINE Emergency Stop
AND NOT   M00811	// W150-1 공압이상
TON       T0882 50	// W150-1 클램프 이상
//   //  공정 상태 표시
; L120
LOAD      F00099
MOV       0 D000800	// W150-1 공정상태
; L121
LOAD      M00802	// W150-1 자동 Mode
AND       M00800	// W150-1 Seleted
AND       F00093
OR        M00803	// W150-1 자동기동
MOV       1 D000800	// W150-1 공정상태
; L123
LOAD      M00801	// W150-1 수동 Mode
MOV       2 D000800	// W150-1 공정상태
; L124
LOAD      M00809	// W150-1 이상
MOV       3 D000800	// W150-1 공정상태
//   // 안전광센서 상태램프
//   // MBR 파트 이상 램프
; L127
LOAD      F00099
MPUSH
AND NOT   P01120	// W150-1 파트1
MOV       0 D000811	// W150-1 파트램프 상태1
MLOAD
AND       P01120	// W150-1 파트1
MOV       1 D000811	// W150-1 파트램프 상태1
MPOP
LOAD      M00814	// W150-1 파트이상
AND NOT   P01120	// W150-1 파트1
LOAD      M0081D	// W150-1 파트센서 체크 이상
AND       P01120	// W150-1 파트1
OR LOAD
AND LOAD
MOV       2 D000811	// W150-1 파트램프 상태1

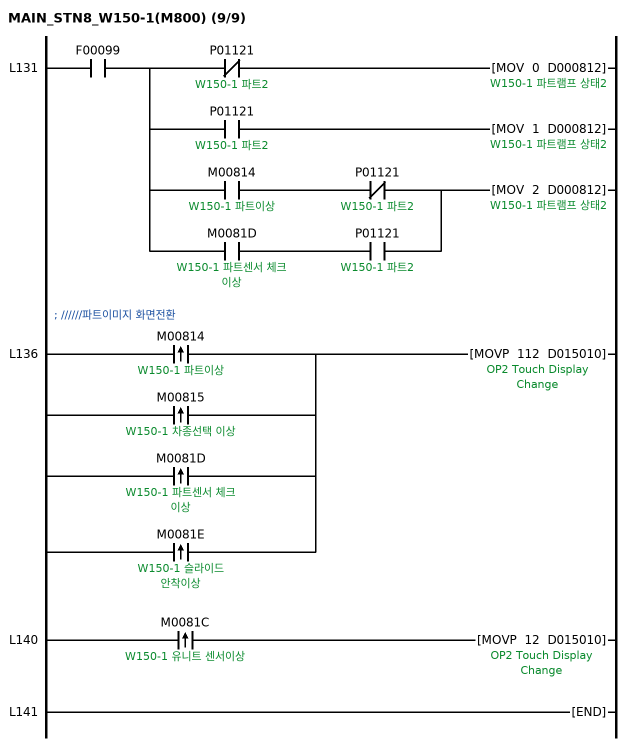
; L131
LOAD      F00099
MPUSH
AND NOT   P01121	// W150-1 파트2
MOV       0 D000812	// W150-1 파트램프 상태2
MLOAD
AND       P01121	// W150-1 파트2
MOV       1 D000812	// W150-1 파트램프 상태2
MPOP
LOAD      M00814	// W150-1 파트이상
AND NOT   P01121	// W150-1 파트2
LOAD      M0081D	// W150-1 파트센서 체크 이상
AND       P01121	// W150-1 파트2
OR LOAD
AND LOAD
MOV       2 D000812	// W150-1 파트램프 상태2
// //////파트이미지 화면전환
; L136
LOADP     M00814	// W150-1 파트이상
ORP       M00815	// W150-1 차종선택 이상
ORP       M0081D	// W150-1 파트센서 체크 이상
ORP       M0081E	// W150-1 슬라이드 안착이상
MOVP      112 D015010	// OP2 Touch Display Change
; L140
LOADP     M0081C	// W150-1 유니트 센서이상
MOVP      12 D015010	// OP2 Touch Display Change
; L141
END

PROGRAM MAIN_STN9_W150-2(M1600) (task: 스캔 프로그램)

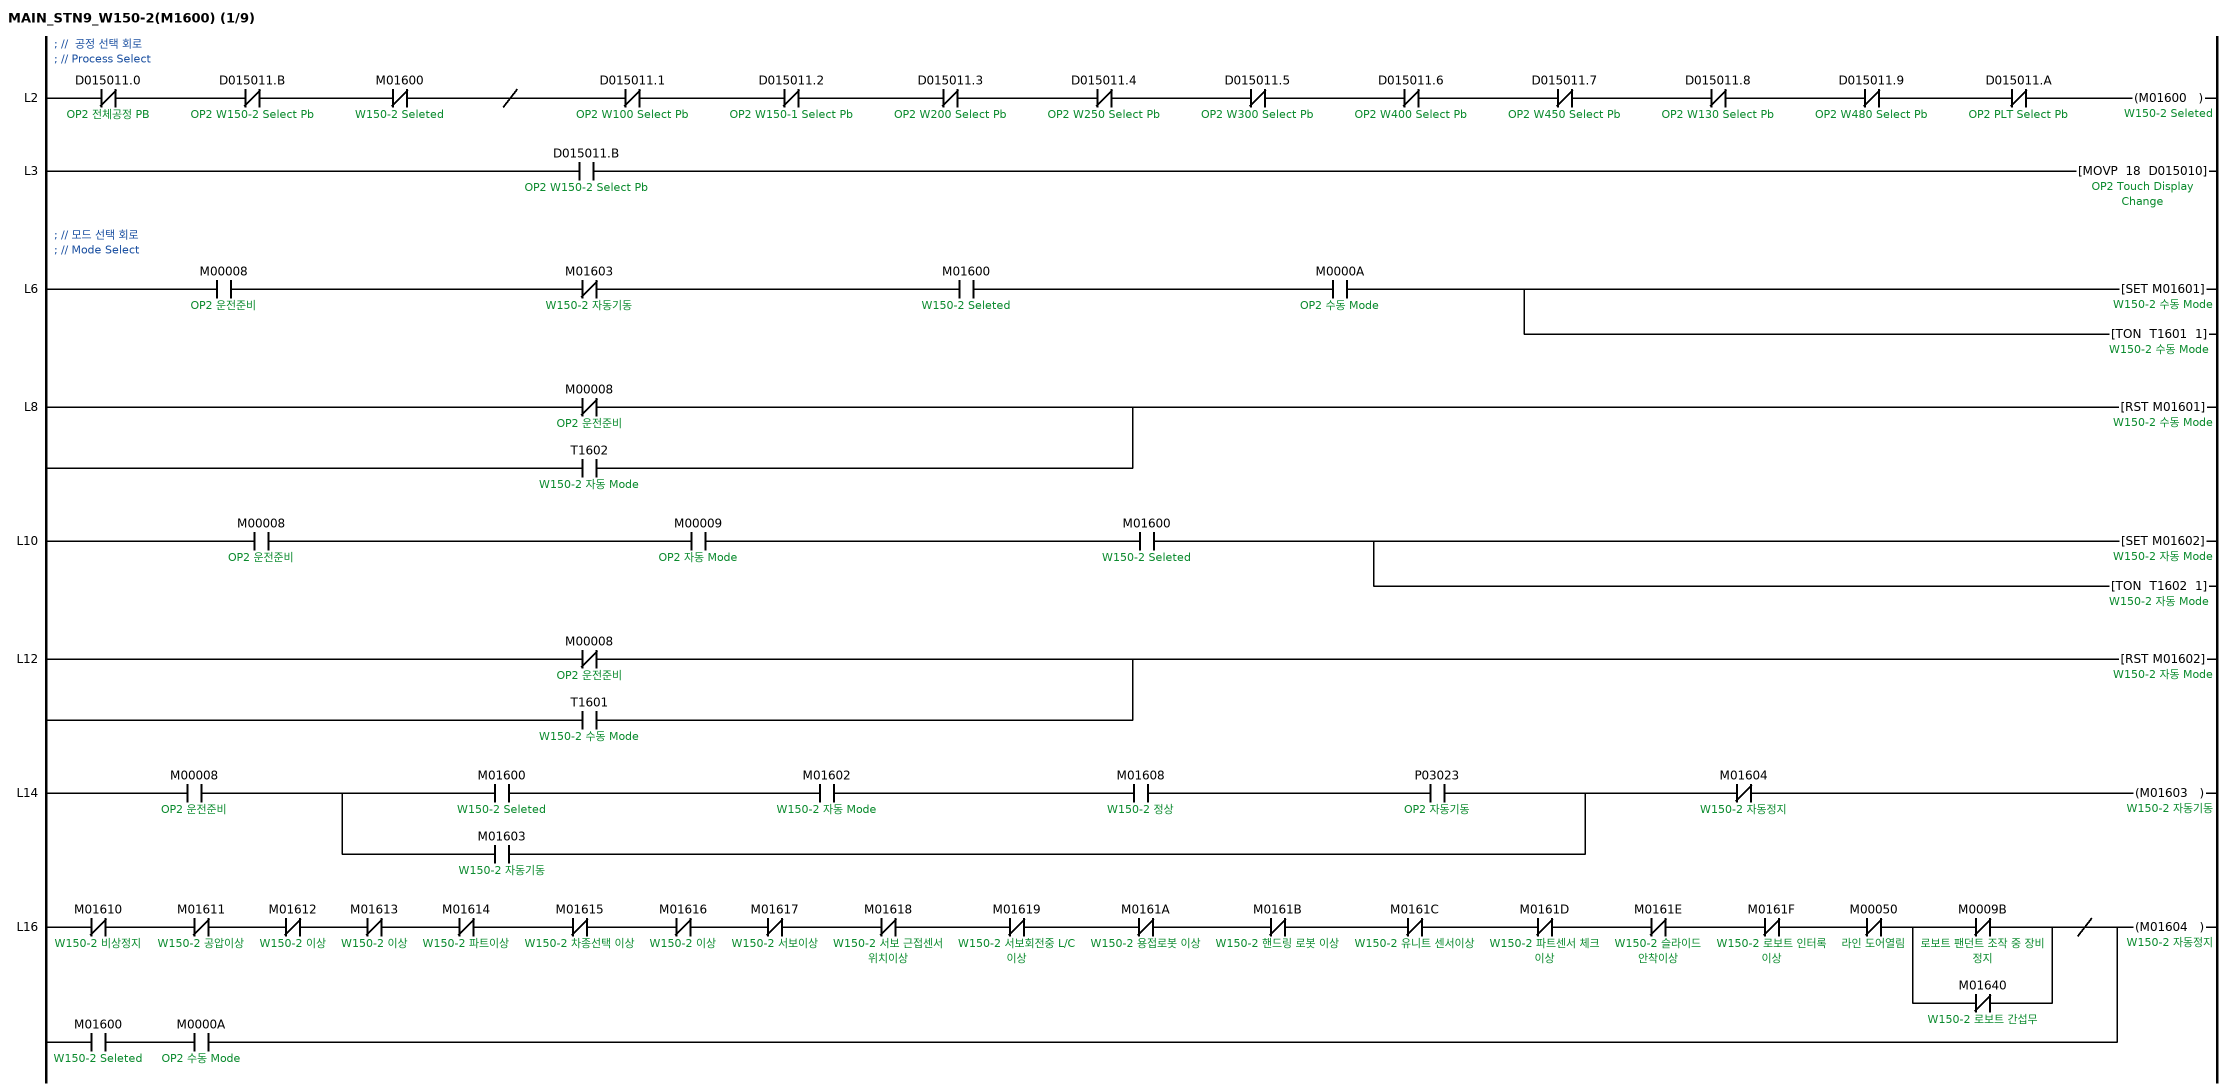
//   //  공정 선택 회로
//   // Process Select
; L2
LOAD NOT  D015011.0	// OP2 전체공정 PB
AND NOT   D015011.B	// OP2 W150-2 Select Pb
AND NOT   M01600	// W150-2 Seleted
NOT
AND NOT   D015011.1	// OP2 W100 Select Pb
AND NOT   D015011.2	// OP2 W150-1 Select Pb
AND NOT   D015011.3	// OP2 W200 Select Pb
AND NOT   D015011.4	// OP2 W250 Select Pb
AND NOT   D015011.5	// OP2 W300 Select Pb
AND NOT   D015011.6	// OP2 W400 Select Pb
AND NOT   D015011.7	// OP2 W450 Select Pb
AND NOT   D015011.8	// OP2 W130 Select Pb
AND NOT   D015011.9	// OP2 W480 Select Pb
AND NOT   D015011.A	// OP2 PLT Select Pb
OUT       M01600	// W150-2 Seleted
; L3
LOAD      D015011.B	// OP2 W150-2 Select Pb
MOVP      18 D015010	// OP2 Touch Display Change
// // 모드 선택 회로
//   // Mode Select
; L6
LOAD      M00008	// OP2 운전준비
AND NOT   M01603	// W150-2 자동기동
AND       M01600	// W150-2 Seleted
AND       M0000A	// OP2 수동 Mode
SET       M01601	// W150-2 수동 Mode
TON       T1601 1	// W150-2 수동 Mode
; L8
LOAD NOT  M00008	// OP2 운전준비
OR        T1602	// W150-2 자동 Mode
RST       M01601	// W150-2 수동 Mode
; L10
LOAD      M00008	// OP2 운전준비
AND       M00009	// OP2 자동 Mode
AND       M01600	// W150-2 Seleted
SET       M01602	// W150-2 자동 Mode
TON       T1602 1	// W150-2 자동 Mode
; L12
LOAD NOT  M00008	// OP2 운전준비
OR        T1601	// W150-2 수동 Mode
RST       M01602	// W150-2 자동 Mode
; L14
LOAD      M00008	// OP2 운전준비
LOAD      M01600	// W150-2 Seleted
AND       M01602	// W150-2 자동 Mode
AND       M01608	// W150-2 정상
AND       P03023	// OP2 자동기동
OR        M01603	// W150-2 자동기동
AND LOAD
AND NOT   M01604	// W150-2 자동정지
OUT       M01603	// W150-2 자동기동
; L16
LOAD NOT  M01610	// W150-2 비상정지
AND NOT   M01611	// W150-2 공압이상
AND NOT   M01612	// W150-2 이상
AND NOT   M01613	// W150-2 이상
AND NOT   M01614	// W150-2 파트이상
AND NOT   M01615	// W150-2 차종선택 이상
AND NOT   M01616	// W150-2 이상
AND NOT   M01617	// W150-2 서보이상
AND NOT   M01618	// W150-2 서보 근접센서 위치이상
AND NOT   M01619	// W150-2 서보회전중 L/C 이상
AND NOT   M0161A	// W150-2 용접로봇 이상
AND NOT   M0161B	// W150-2 핸드링 로봇 이상
AND NOT   M0161C	// W150-2 유니트 센서이상
AND NOT   M0161D	// W150-2 파트센서 체크 이상
AND NOT   M0161E	// W150-2 슬라이드 안착이상
AND NOT   M0161F	// W150-2 로보트 인터록 이상
AND NOT   M00050	// 라인 도어열림
LOAD NOT  M0009B	// 로보트 팬던트 조작 중 장비 정지
OR NOT    M01640	// W150-2 로보트 간섭무
AND LOAD
NOT
LOAD      M01600	// W150-2 Seleted
AND       M0000A	// OP2 수동 Mode
OR LOAD
OUT       M01604	// W150-2 자동정지

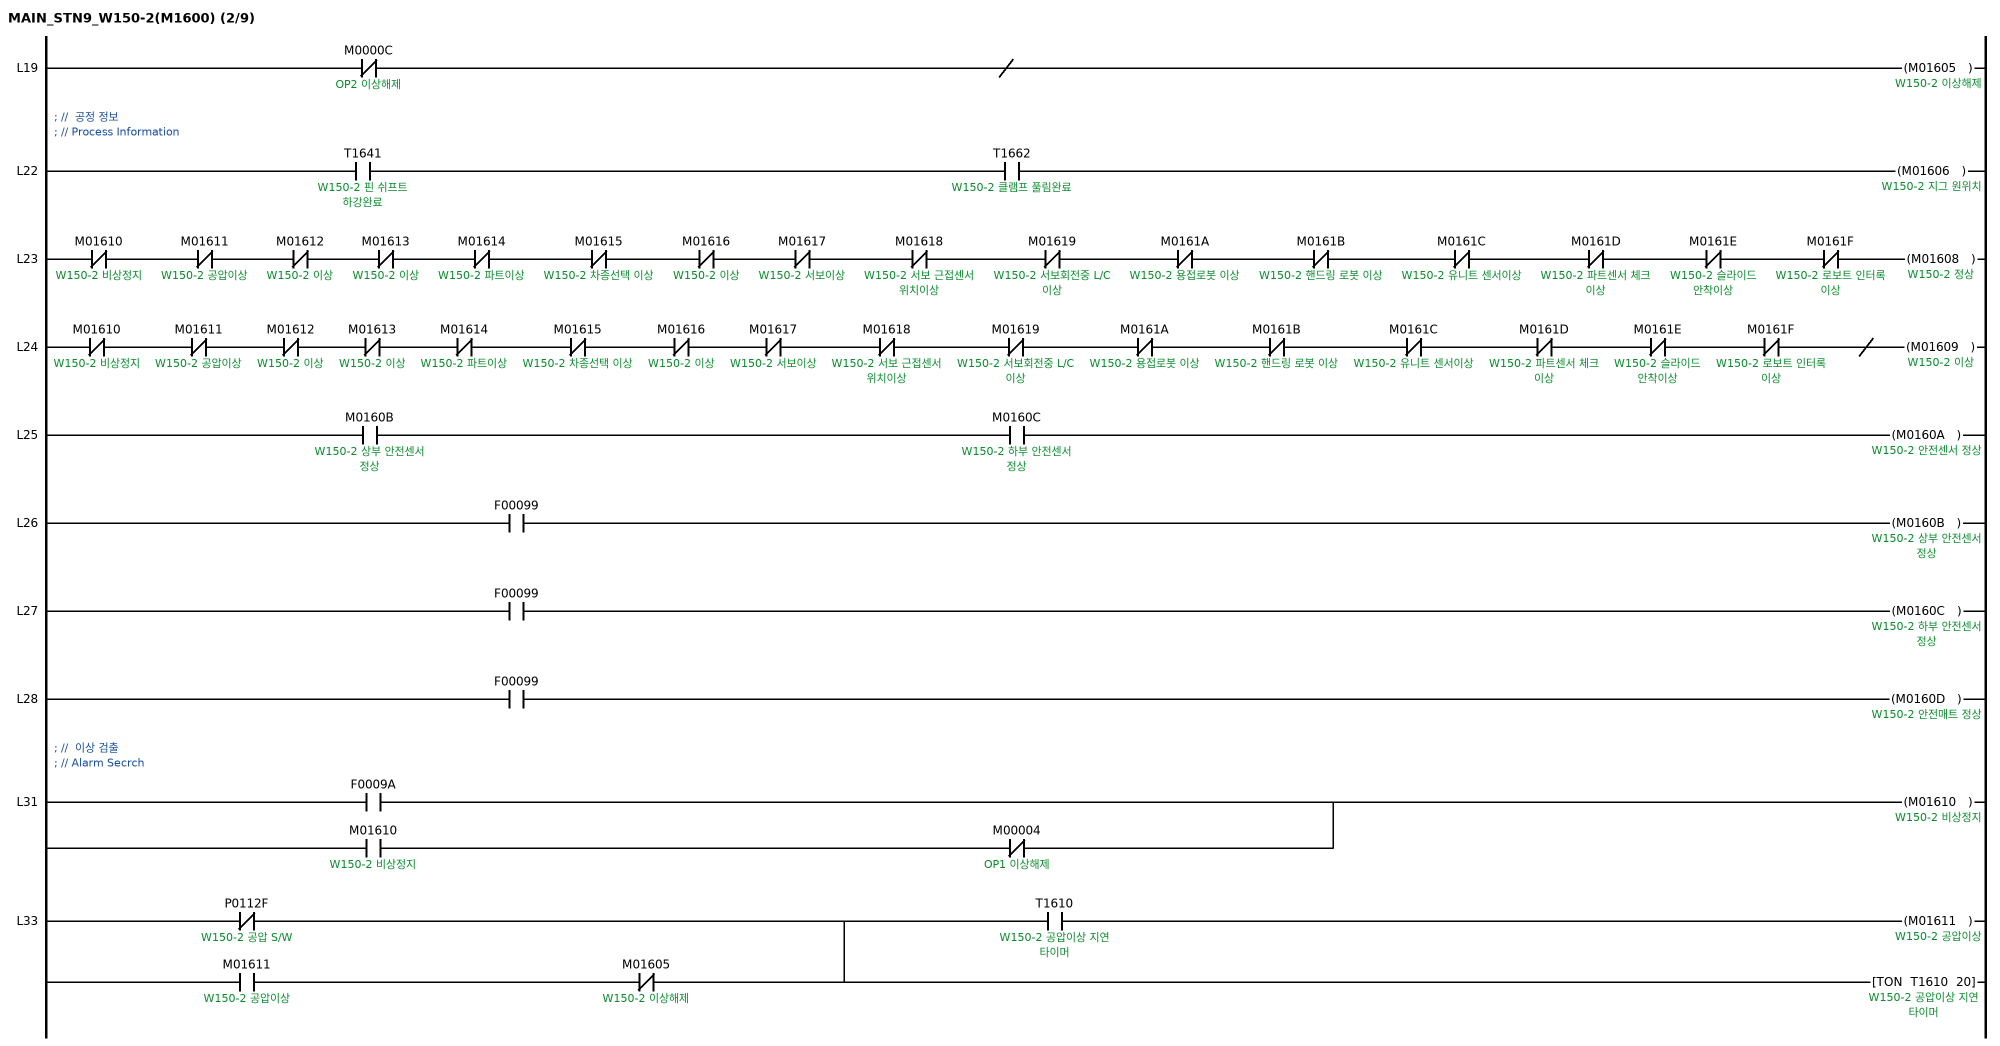
; L19
LOAD NOT  M0000C	// OP2 이상해제
NOT
OUT       M01605	// W150-2 이상해제
//   //  공정 정보
//   // Process Information
; L22
LOAD      T1641	// W150-2 핀 쉬프트 하강완료
AND       T1662	// W150-2 클램프 풀림완료
OUT       M01606	// W150-2 지그 원위치
; L23
LOAD NOT  M01610	// W150-2 비상정지
AND NOT   M01611	// W150-2 공압이상
AND NOT   M01612	// W150-2 이상
AND NOT   M01613	// W150-2 이상
AND NOT   M01614	// W150-2 파트이상
AND NOT   M01615	// W150-2 차종선택 이상
AND NOT   M01616	// W150-2 이상
AND NOT   M01617	// W150-2 서보이상
AND NOT   M01618	// W150-2 서보 근접센서 위치이상
AND NOT   M01619	// W150-2 서보회전중 L/C 이상
AND NOT   M0161A	// W150-2 용접로봇 이상
AND NOT   M0161B	// W150-2 핸드링 로봇 이상
AND NOT   M0161C	// W150-2 유니트 센서이상
AND NOT   M0161D	// W150-2 파트센서 체크 이상
AND NOT   M0161E	// W150-2 슬라이드 안착이상
AND NOT   M0161F	// W150-2 로보트 인터록 이상
OUT       M01608	// W150-2 정상
; L24
LOAD NOT  M01610	// W150-2 비상정지
AND NOT   M01611	// W150-2 공압이상
AND NOT   M01612	// W150-2 이상
AND NOT   M01613	// W150-2 이상
AND NOT   M01614	// W150-2 파트이상
AND NOT   M01615	// W150-2 차종선택 이상
AND NOT   M01616	// W150-2 이상
AND NOT   M01617	// W150-2 서보이상
AND NOT   M01618	// W150-2 서보 근접센서 위치이상
AND NOT   M01619	// W150-2 서보회전중 L/C 이상
AND NOT   M0161A	// W150-2 용접로봇 이상
AND NOT   M0161B	// W150-2 핸드링 로봇 이상
AND NOT   M0161C	// W150-2 유니트 센서이상
AND NOT   M0161D	// W150-2 파트센서 체크 이상
AND NOT   M0161E	// W150-2 슬라이드 안착이상
AND NOT   M0161F	// W150-2 로보트 인터록 이상
NOT
OUT       M01609	// W150-2 이상
; L25
LOAD      M0160B	// W150-2 상부 안전센서 정상
AND       M0160C	// W150-2 하부 안전센서 정상
OUT       M0160A	// W150-2 안전센서 정상
; L26
LOAD      F00099
OUT       M0160B	// W150-2 상부 안전센서 정상
; L27
LOAD      F00099
OUT       M0160C	// W150-2 하부 안전센서 정상
; L28
LOAD      F00099
OUT       M0160D	// W150-2 안전매트 정상
//   //  이상 검출
//   // Alarm Secrch
; L31
LOAD      F0009A
LOAD      M01610	// W150-2 비상정지
AND NOT   M00004	// OP1 이상해제
OR LOAD
OUT       M01610	// W150-2 비상정지
; L33
LOAD NOT  P0112F	// W150-2 공압 S/W
LOAD      M01611	// W150-2 공압이상
AND NOT   M01605	// W150-2 이상해제
OR LOAD
MPUSH
AND       T1610	// W150-2 공압이상 지연 타이머
OUT       M01611	// W150-2 공압이상
MPOP
TON       T1610 20	// W150-2 공압이상 지연 타이머

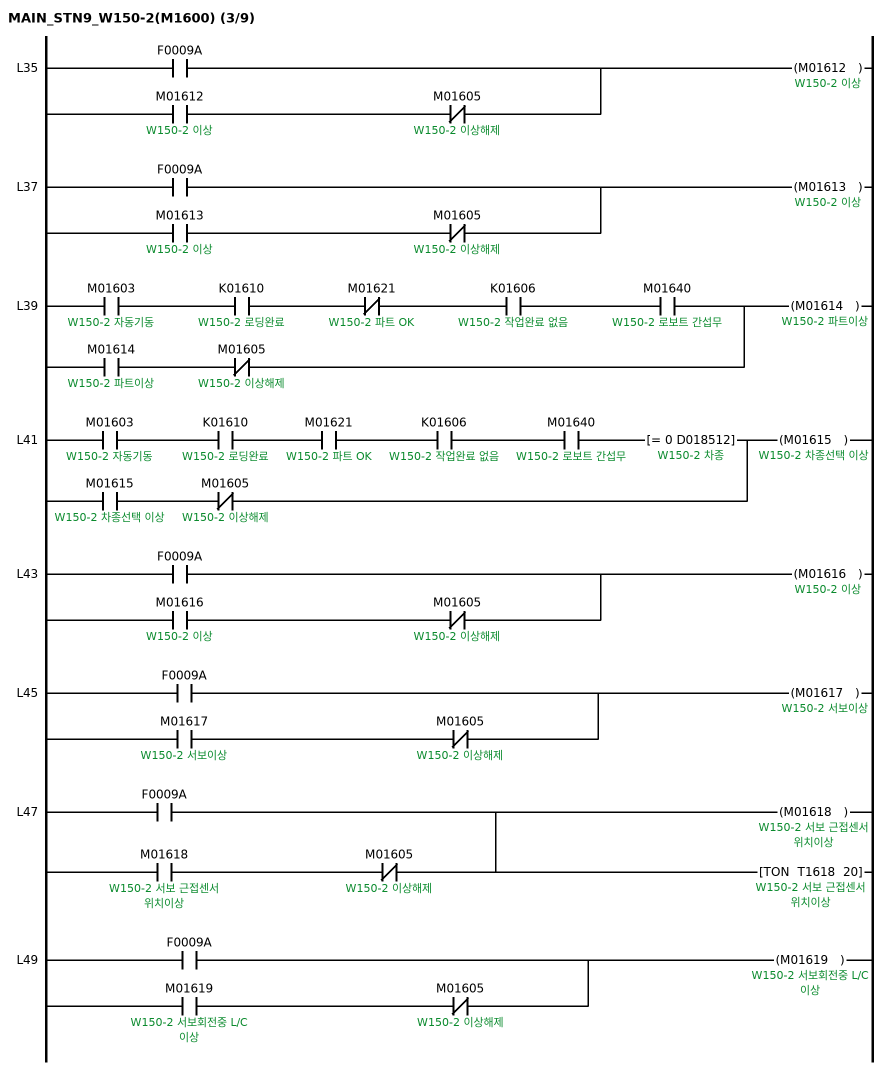
; L35
LOAD      F0009A
LOAD      M01612	// W150-2 이상
AND NOT   M01605	// W150-2 이상해제
OR LOAD
OUT       M01612	// W150-2 이상
; L37
LOAD      F0009A
LOAD      M01613	// W150-2 이상
AND NOT   M01605	// W150-2 이상해제
OR LOAD
OUT       M01613	// W150-2 이상
; L39
LOAD      M01603	// W150-2 자동기동
AND       K01610	// W150-2 로딩완료
AND NOT   M01621	// W150-2 파트 OK
AND       K01606	// W150-2 작업완료 없음
AND       M01640	// W150-2 로보트 간섭무
LOAD      M01614	// W150-2 파트이상
AND NOT   M01605	// W150-2 이상해제
OR LOAD
OUT       M01614	// W150-2 파트이상
; L41
LOAD      M01603	// W150-2 자동기동
AND       K01610	// W150-2 로딩완료
AND       M01621	// W150-2 파트 OK
AND       K01606	// W150-2 작업완료 없음
AND       M01640	// W150-2 로보트 간섭무
AND=      0 D018512	// W150-2 차종
LOAD      M01615	// W150-2 차종선택 이상
AND NOT   M01605	// W150-2 이상해제
OR LOAD
OUT       M01615	// W150-2 차종선택 이상
; L43
LOAD      F0009A
LOAD      M01616	// W150-2 이상
AND NOT   M01605	// W150-2 이상해제
OR LOAD
OUT       M01616	// W150-2 이상
; L45
LOAD      F0009A
LOAD      M01617	// W150-2 서보이상
AND NOT   M01605	// W150-2 이상해제
OR LOAD
OUT       M01617	// W150-2 서보이상
; L47
LOAD      F0009A
LOAD      M01618	// W150-2 서보 근접센서 위치이상
AND NOT   M01605	// W150-2 이상해제
OR LOAD
OUT       M01618	// W150-2 서보 근접센서 위치이상
TON       T1618 20	// W150-2 서보 근접센서 위치이상
; L49
LOAD      F0009A
LOAD      M01619	// W150-2 서보회전중 L/C 이상
AND NOT   M01605	// W150-2 이상해제
OR LOAD
OUT       M01619	// W150-2 서보회전중 L/C 이상

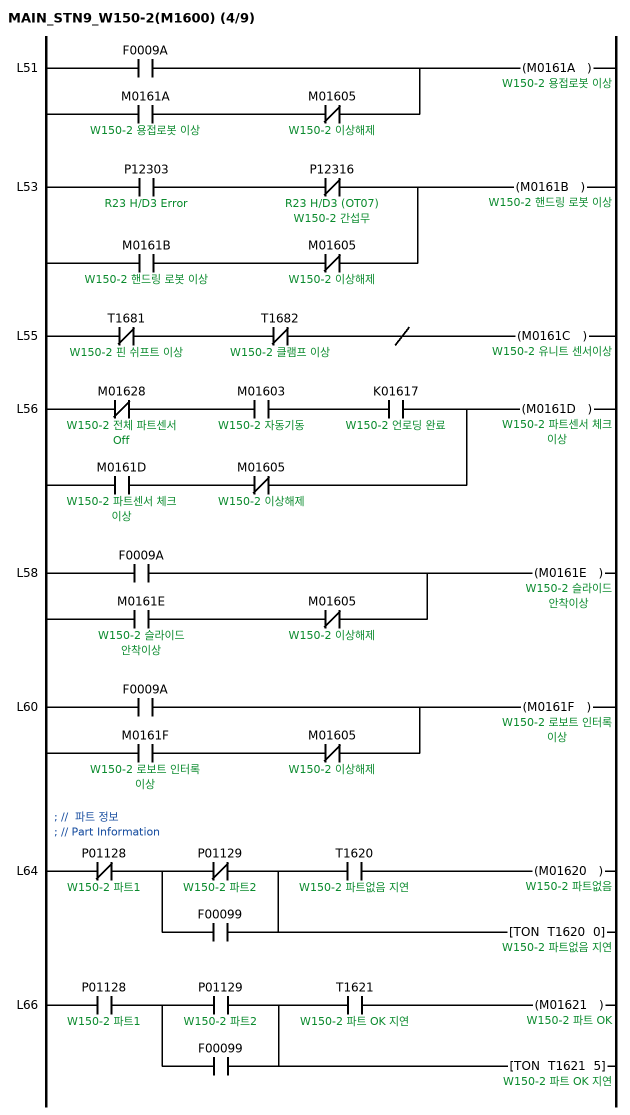
; L51
LOAD      F0009A
LOAD      M0161A	// W150-2 용접로봇 이상
AND NOT   M01605	// W150-2 이상해제
OR LOAD
OUT       M0161A	// W150-2 용접로봇 이상
; L53
LOAD      P12303	// R23 H/D3 Error
AND NOT   P12316	// R23 H/D3 (OT07) W150-2 간섭무
LOAD      M0161B	// W150-2 핸드링 로봇 이상
AND NOT   M01605	// W150-2 이상해제
OR LOAD
OUT       M0161B	// W150-2 핸드링 로봇 이상
; L55
LOAD NOT  T1681	// W150-2 핀 쉬프트 이상
AND NOT   T1682	// W150-2 클램프 이상
NOT
OUT       M0161C	// W150-2 유니트 센서이상
; L56
LOAD NOT  M01628	// W150-2 전체 파트센서 Off
AND       M01603	// W150-2 자동기동
AND       K01617	// W150-2 언로딩 완료
LOAD      M0161D	// W150-2 파트센서 체크 이상
AND NOT   M01605	// W150-2 이상해제
OR LOAD
OUT       M0161D	// W150-2 파트센서 체크 이상
; L58
LOAD      F0009A
LOAD      M0161E	// W150-2 슬라이드 안착이상
AND NOT   M01605	// W150-2 이상해제
OR LOAD
OUT       M0161E	// W150-2 슬라이드 안착이상
; L60
LOAD      F0009A
LOAD      M0161F	// W150-2 로보트 인터록 이상
AND NOT   M01605	// W150-2 이상해제
OR LOAD
OUT       M0161F	// W150-2 로보트 인터록 이상
//   //  파트 정보
//   // Part Information
; L64
LOAD NOT  P01128	// W150-2 파트1
LOAD NOT  P01129	// W150-2 파트2
OR        F00099
AND LOAD
MPUSH
AND       T1620	// W150-2 파트없음 지연
OUT       M01620	// W150-2 파트없음
MPOP
TON       T1620 0	// W150-2 파트없음 지연
; L66
LOAD      P01128	// W150-2 파트1
LOAD      P01129	// W150-2 파트2
OR        F00099
AND LOAD
MPUSH
AND       T1621	// W150-2 파트 OK 지연
OUT       M01621	// W150-2 파트 OK
MPOP
TON       T1621 5	// W150-2 파트 OK 지연

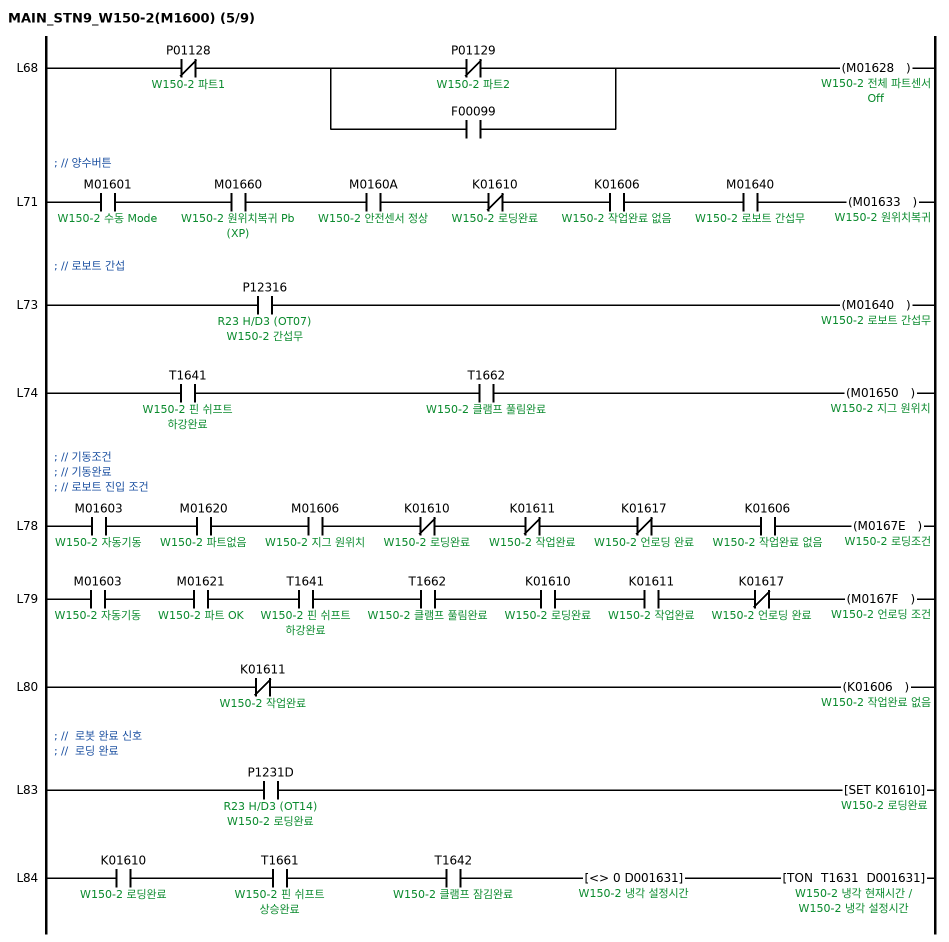
; L68
LOAD NOT  P01128	// W150-2 파트1
LOAD NOT  P01129	// W150-2 파트2
OR        F00099
AND LOAD
OUT       M01628	// W150-2 전체 파트센서 Off
//   // 양수버튼
; L71
LOAD      M01601	// W150-2 수동 Mode
AND       M01660	// W150-2 원위치복귀 Pb (XP)
AND       M0160A	// W150-2 안전센서 정상
AND NOT   K01610	// W150-2 로딩완료
AND       K01606	// W150-2 작업완료 없음
AND       M01640	// W150-2 로보트 간섭무
OUT       M01633	// W150-2 원위치복귀
//   // 로보트 간섭
; L73
LOAD      P12316	// R23 H/D3 (OT07) W150-2 간섭무
OUT       M01640	// W150-2 로보트 간섭무
; L74
LOAD      T1641	// W150-2 핀 쉬프트 하강완료
AND       T1662	// W150-2 클램프 풀림완료
OUT       M01650	// W150-2 지그 원위치
//   // 기동조건
//   // 기동완료
//   // 로보트 진입 조건
; L78
LOAD      M01603	// W150-2 자동기동
AND       M01620	// W150-2 파트없음
AND       M01606	// W150-2 지그 원위치
AND NOT   K01610	// W150-2 로딩완료
AND NOT   K01611	// W150-2 작업완료
AND NOT   K01617	// W150-2 언로딩 완료
AND       K01606	// W150-2 작업완료 없음
OUT       M0167E	// W150-2 로딩조건
; L79
LOAD      M01603	// W150-2 자동기동
AND       M01621	// W150-2 파트 OK
AND       T1641	// W150-2 핀 쉬프트 하강완료
AND       T1662	// W150-2 클램프 풀림완료
AND       K01610	// W150-2 로딩완료
AND       K01611	// W150-2 작업완료
AND NOT   K01617	// W150-2 언로딩 완료
OUT       M0167F	// W150-2 언로딩 조건
; L80
LOAD NOT  K01611	// W150-2 작업완료
OUT       K01606	// W150-2 작업완료 없음
//   //  로봇 완료 신호
//   //  로딩 완료
; L83
LOAD      P1231D	// R23 H/D3 (OT14) W150-2 로딩완료
SET       K01610	// W150-2 로딩완료
; L84
LOAD      K01610	// W150-2 로딩완료
AND       T1661	// W150-2 핀 쉬프트 상승완료
AND       T1642	// W150-2 클램프 잠김완료
AND<>     0 D001631	// W150-2 냉각 설정시간
TON       T1631 D001631	// W150-2 냉각 현재시간 / W150-2 냉각 설정시간

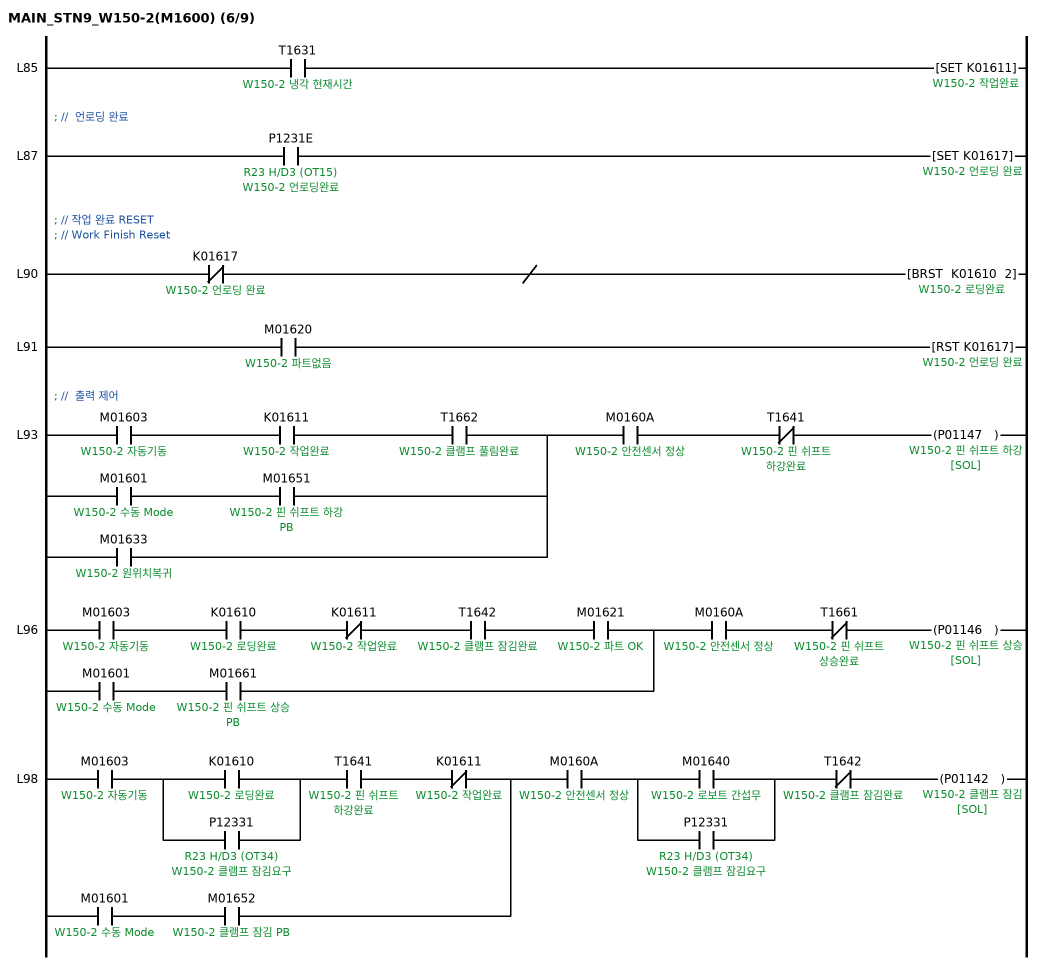
; L85
LOAD      T1631	// W150-2 냉각 현재시간
SET       K01611	// W150-2 작업완료
//   //  언로딩 완료
; L87
LOAD      P1231E	// R23 H/D3 (OT15) W150-2 언로딩완료
SET       K01617	// W150-2 언로딩 완료
//     // 작업 완료 RESET
//   // Work Finish Reset
; L90
LOAD NOT  K01617	// W150-2 언로딩 완료
NOT
BRST      K01610 2	// W150-2 로딩완료
; L91
LOAD      M01620	// W150-2 파트없음
RST       K01617	// W150-2 언로딩 완료
//     //  출력 제어
; L93
LOAD      M01603	// W150-2 자동기동
AND       K01611	// W150-2 작업완료
AND       T1662	// W150-2 클램프 풀림완료
LOAD      M01601	// W150-2 수동 Mode
AND       M01651	// W150-2 핀 쉬프트 하강 PB
OR LOAD
OR        M01633	// W150-2 원위치복귀
AND       M0160A	// W150-2 안전센서 정상
AND NOT   T1641	// W150-2 핀 쉬프트 하강완료
OUT       P01147	// W150-2 핀 쉬프트 하강 [SOL]
; L96
LOAD      M01603	// W150-2 자동기동
AND       K01610	// W150-2 로딩완료
AND NOT   K01611	// W150-2 작업완료
AND       T1642	// W150-2 클램프 잠김완료
AND       M01621	// W150-2 파트 OK
LOAD      M01601	// W150-2 수동 Mode
AND       M01661	// W150-2 핀 쉬프트 상승 PB
OR LOAD
AND       M0160A	// W150-2 안전센서 정상
AND NOT   T1661	// W150-2 핀 쉬프트 상승완료
OUT       P01146	// W150-2 핀 쉬프트 상승 [SOL]
; L98
LOAD      M01603	// W150-2 자동기동
LOAD      K01610	// W150-2 로딩완료
OR        P12331	// R23 H/D3 (OT34) W150-2 클램프 잠김요구
AND LOAD
AND       T1641	// W150-2 핀 쉬프트 하강완료
AND NOT   K01611	// W150-2 작업완료
LOAD      M01601	// W150-2 수동 Mode
AND       M01652	// W150-2 클램프 잠김 PB
OR LOAD
AND       M0160A	// W150-2 안전센서 정상
LOAD      M01640	// W150-2 로보트 간섭무
OR        P12331	// R23 H/D3 (OT34) W150-2 클램프 잠김요구
AND LOAD
AND NOT   T1642	// W150-2 클램프 잠김완료
OUT       P01142	// W150-2 클램프 잠김 [SOL]

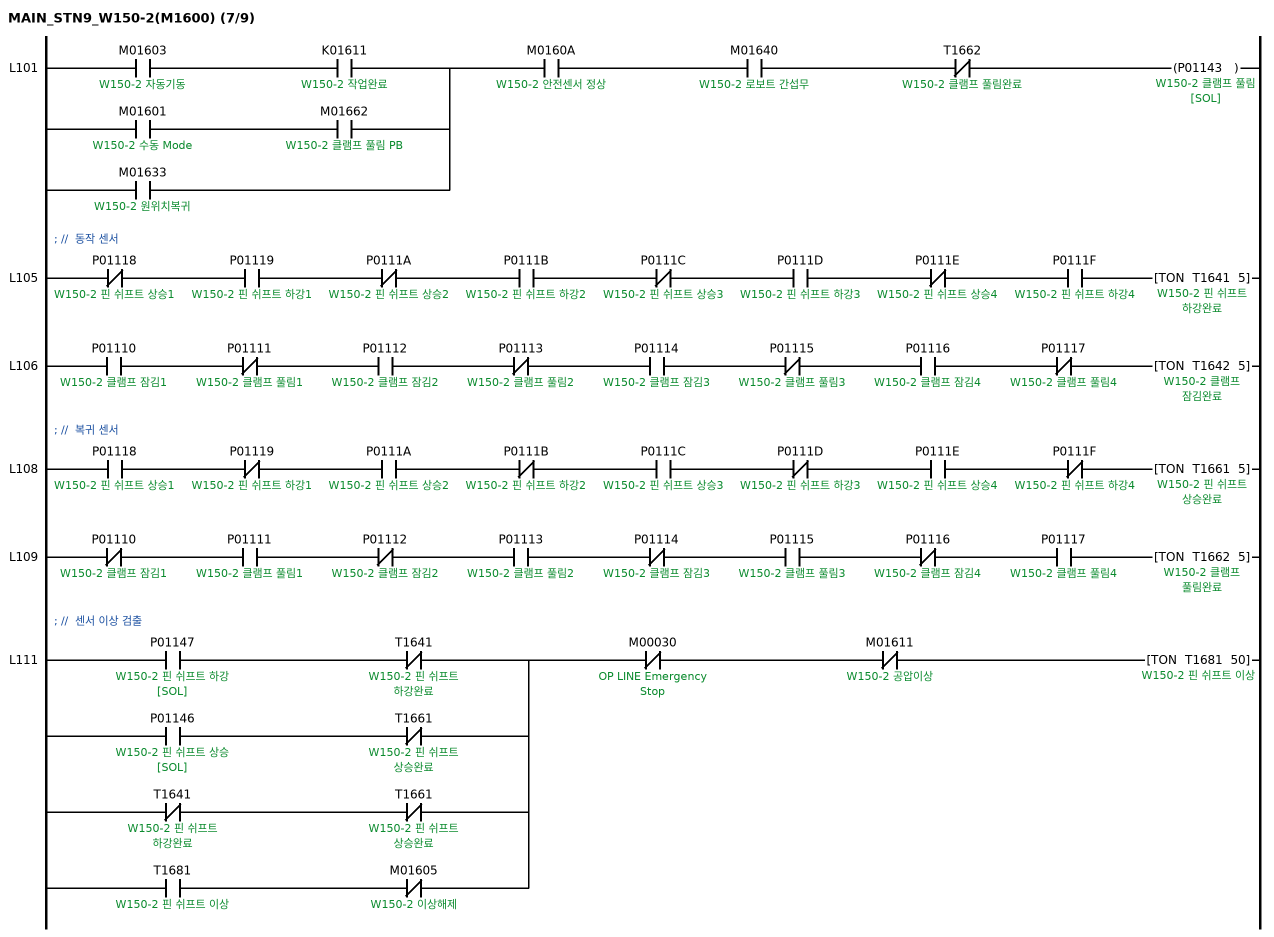
; L101
LOAD      M01603	// W150-2 자동기동
AND       K01611	// W150-2 작업완료
LOAD      M01601	// W150-2 수동 Mode
AND       M01662	// W150-2 클램프 풀림 PB
OR LOAD
OR        M01633	// W150-2 원위치복귀
AND       M0160A	// W150-2 안전센서 정상
AND       M01640	// W150-2 로보트 간섭무
AND NOT   T1662	// W150-2 클램프 풀림완료
OUT       P01143	// W150-2 클램프 풀림 [SOL]
//   //  동작 센서
; L105
LOAD NOT  P01118	// W150-2 핀 쉬프트 상승1
AND       P01119	// W150-2 핀 쉬프트 하강1
AND NOT   P0111A	// W150-2 핀 쉬프트 상승2
AND       P0111B	// W150-2 핀 쉬프트 하강2
AND NOT   P0111C	// W150-2 핀 쉬프트 상승3
AND       P0111D	// W150-2 핀 쉬프트 하강3
AND NOT   P0111E	// W150-2 핀 쉬프트 상승4
AND       P0111F	// W150-2 핀 쉬프트 하강4
TON       T1641 5	// W150-2 핀 쉬프트 하강완료
; L106
LOAD      P01110	// W150-2 클램프 잠김1
AND NOT   P01111	// W150-2 클램프 풀림1
AND       P01112	// W150-2 클램프 잠김2
AND NOT   P01113	// W150-2 클램프 풀림2
AND       P01114	// W150-2 클램프 잠김3
AND NOT   P01115	// W150-2 클램프 풀림3
AND       P01116	// W150-2 클램프 잠김4
AND NOT   P01117	// W150-2 클램프 풀림4
TON       T1642 5	// W150-2 클램프 잠김완료
//   //  복귀 센서
; L108
LOAD      P01118	// W150-2 핀 쉬프트 상승1
AND NOT   P01119	// W150-2 핀 쉬프트 하강1
AND       P0111A	// W150-2 핀 쉬프트 상승2
AND NOT   P0111B	// W150-2 핀 쉬프트 하강2
AND       P0111C	// W150-2 핀 쉬프트 상승3
AND NOT   P0111D	// W150-2 핀 쉬프트 하강3
AND       P0111E	// W150-2 핀 쉬프트 상승4
AND NOT   P0111F	// W150-2 핀 쉬프트 하강4
TON       T1661 5	// W150-2 핀 쉬프트 상승완료
; L109
LOAD NOT  P01110	// W150-2 클램프 잠김1
AND       P01111	// W150-2 클램프 풀림1
AND NOT   P01112	// W150-2 클램프 잠김2
AND       P01113	// W150-2 클램프 풀림2
AND NOT   P01114	// W150-2 클램프 잠김3
AND       P01115	// W150-2 클램프 풀림3
AND NOT   P01116	// W150-2 클램프 잠김4
AND       P01117	// W150-2 클램프 풀림4
TON       T1662 5	// W150-2 클램프 풀림완료
//     //  센서 이상 검출
; L111
LOAD      P01147	// W150-2 핀 쉬프트 하강 [SOL]
AND NOT   T1641	// W150-2 핀 쉬프트 하강완료
LOAD      P01146	// W150-2 핀 쉬프트 상승 [SOL]
AND NOT   T1661	// W150-2 핀 쉬프트 상승완료
OR LOAD
LOAD NOT  T1641	// W150-2 핀 쉬프트 하강완료
AND NOT   T1661	// W150-2 핀 쉬프트 상승완료
OR LOAD
LOAD      T1681	// W150-2 핀 쉬프트 이상
AND NOT   M01605	// W150-2 이상해제
OR LOAD
AND NOT   M00030	// OP LINE Emergency Stop
AND NOT   M01611	// W150-2 공압이상
TON       T1681 50	// W150-2 핀 쉬프트 이상

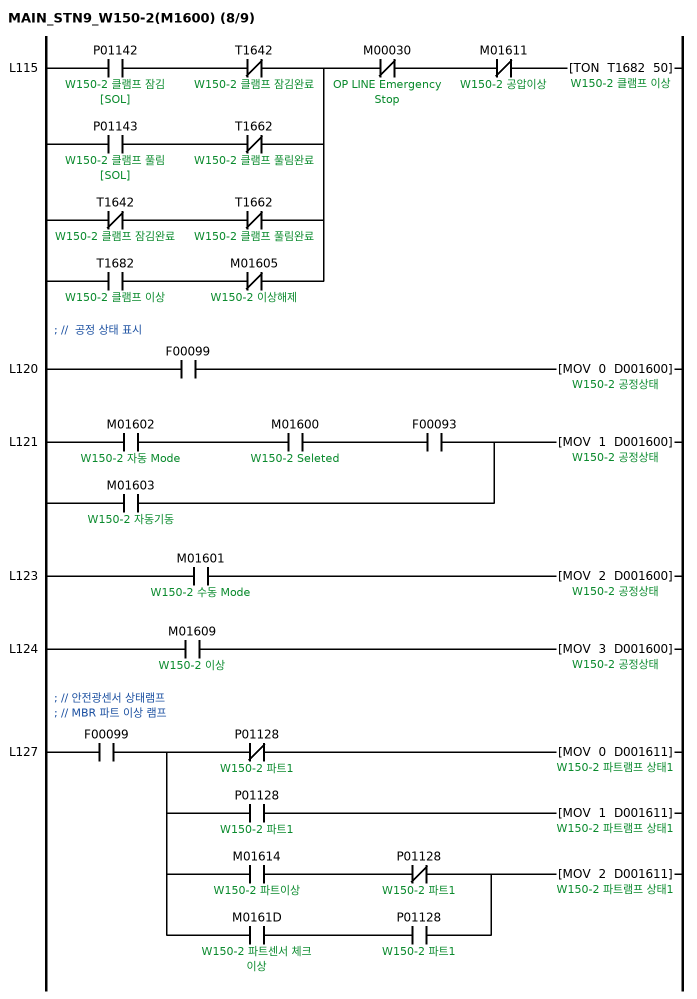
; L115
LOAD      P01142	// W150-2 클램프 잠김 [SOL]
AND NOT   T1642	// W150-2 클램프 잠김완료
LOAD      P01143	// W150-2 클램프 풀림 [SOL]
AND NOT   T1662	// W150-2 클램프 풀림완료
OR LOAD
LOAD NOT  T1642	// W150-2 클램프 잠김완료
AND NOT   T1662	// W150-2 클램프 풀림완료
OR LOAD
LOAD      T1682	// W150-2 클램프 이상
AND NOT   M01605	// W150-2 이상해제
OR LOAD
AND NOT   M00030	// OP LINE Emergency Stop
AND NOT   M01611	// W150-2 공압이상
TON       T1682 50	// W150-2 클램프 이상
//   //  공정 상태 표시
; L120
LOAD      F00099
MOV       0 D001600	// W150-2 공정상태
; L121
LOAD      M01602	// W150-2 자동 Mode
AND       M01600	// W150-2 Seleted
AND       F00093
OR        M01603	// W150-2 자동기동
MOV       1 D001600	// W150-2 공정상태
; L123
LOAD      M01601	// W150-2 수동 Mode
MOV       2 D001600	// W150-2 공정상태
; L124
LOAD      M01609	// W150-2 이상
MOV       3 D001600	// W150-2 공정상태
//   // 안전광센서 상태램프
//   // MBR 파트 이상 램프
; L127
LOAD      F00099
MPUSH
AND NOT   P01128	// W150-2 파트1
MOV       0 D001611	// W150-2 파트램프 상태1
MLOAD
AND       P01128	// W150-2 파트1
MOV       1 D001611	// W150-2 파트램프 상태1
MPOP
LOAD      M01614	// W150-2 파트이상
AND NOT   P01128	// W150-2 파트1
LOAD      M0161D	// W150-2 파트센서 체크 이상
AND       P01128	// W150-2 파트1
OR LOAD
AND LOAD
MOV       2 D001611	// W150-2 파트램프 상태1

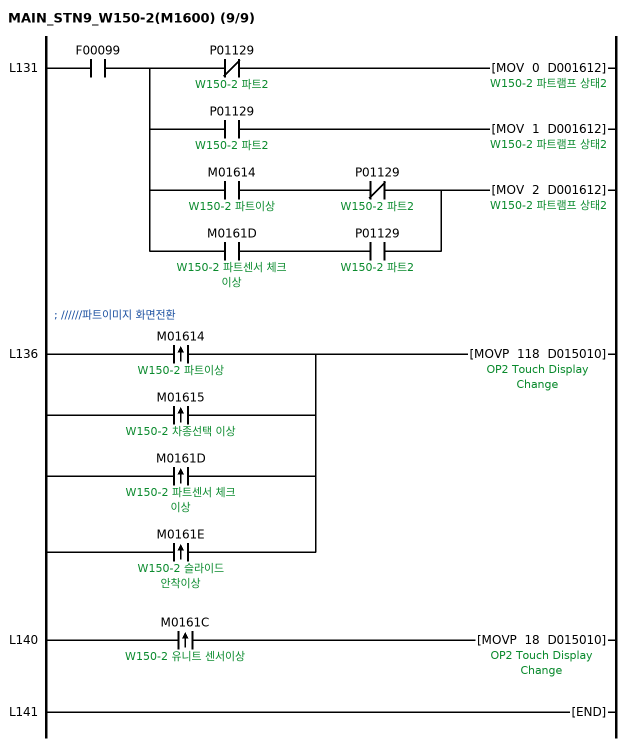
; L131
LOAD      F00099
MPUSH
AND NOT   P01129	// W150-2 파트2
MOV       0 D001612	// W150-2 파트램프 상태2
MLOAD
AND       P01129	// W150-2 파트2
MOV       1 D001612	// W150-2 파트램프 상태2
MPOP
LOAD      M01614	// W150-2 파트이상
AND NOT   P01129	// W150-2 파트2
LOAD      M0161D	// W150-2 파트센서 체크 이상
AND       P01129	// W150-2 파트2
OR LOAD
AND LOAD
MOV       2 D001612	// W150-2 파트램프 상태2
// //////파트이미지 화면전환
; L136
LOADP     M01614	// W150-2 파트이상
ORP       M01615	// W150-2 차종선택 이상
ORP       M0161D	// W150-2 파트센서 체크 이상
ORP       M0161E	// W150-2 슬라이드 안착이상
MOVP      118 D015010	// OP2 Touch Display Change
; L140
LOADP     M0161C	// W150-2 유니트 센서이상
MOVP      18 D015010	// OP2 Touch Display Change
; L141
END

PROGRAM MAIN_STN10_W200(M900) (task: 스캔 프로그램)

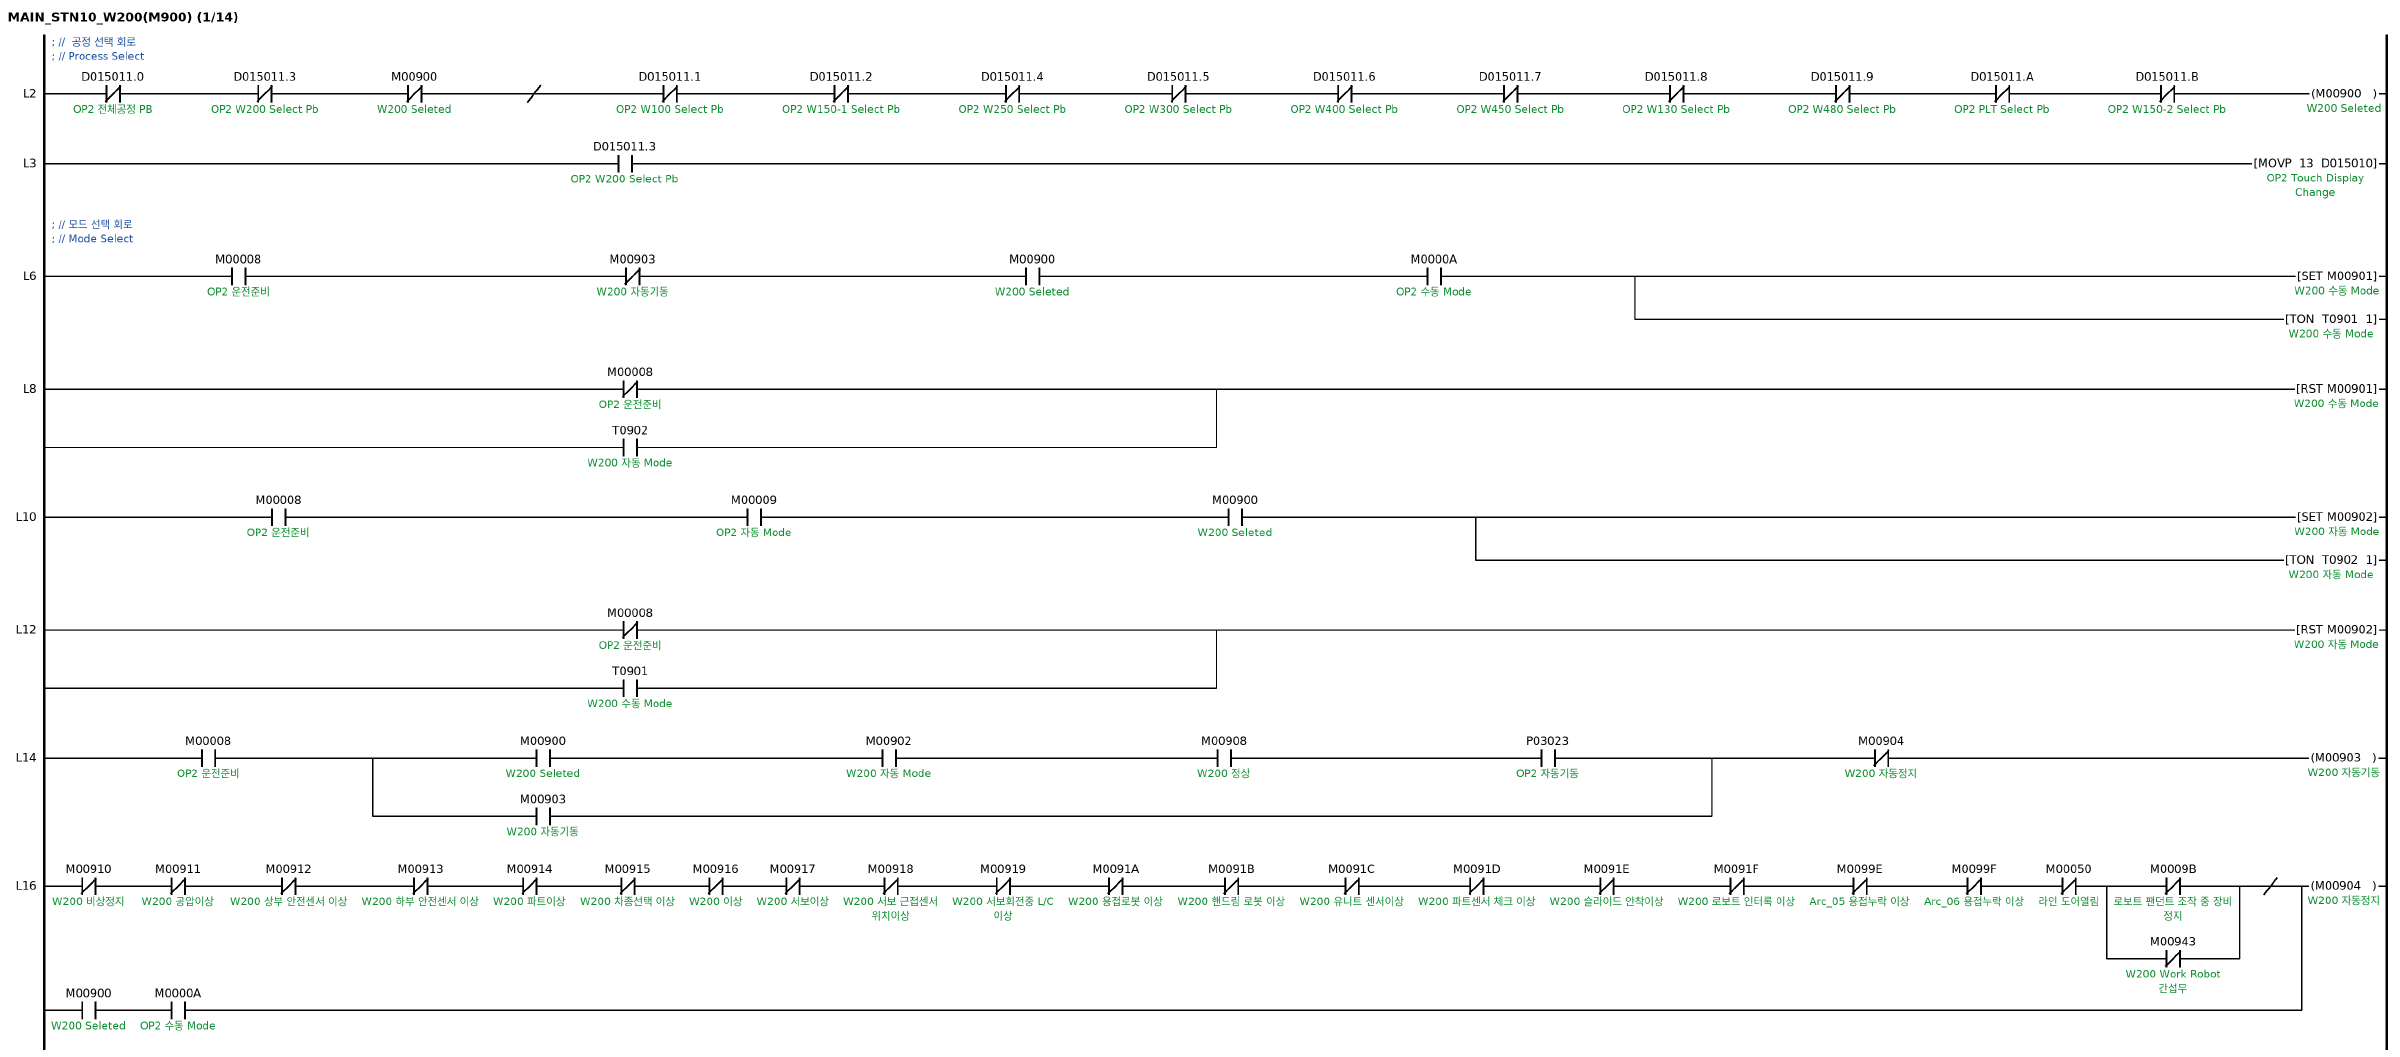
//   //  공정 선택 회로
//   // Process Select
; L2
LOAD NOT  D015011.0	// OP2 전체공정 PB
AND NOT   D015011.3	// OP2 W200 Select Pb
AND NOT   M00900	// W200 Seleted
NOT
AND NOT   D015011.1	// OP2 W100 Select Pb
AND NOT   D015011.2	// OP2 W150-1 Select Pb
AND NOT   D015011.4	// OP2 W250 Select Pb
AND NOT   D015011.5	// OP2 W300 Select Pb
AND NOT   D015011.6	// OP2 W400 Select Pb
AND NOT   D015011.7	// OP2 W450 Select Pb
AND NOT   D015011.8	// OP2 W130 Select Pb
AND NOT   D015011.9	// OP2 W480 Select Pb
AND NOT   D015011.A	// OP2 PLT Select Pb
AND NOT   D015011.B	// OP2 W150-2 Select Pb
OUT       M00900	// W200 Seleted
; L3
LOAD      D015011.3	// OP2 W200 Select Pb
MOVP      13 D015010	// OP2 Touch Display Change
// // 모드 선택 회로
//   // Mode Select
; L6
LOAD      M00008	// OP2 운전준비
AND NOT   M00903	// W200 자동기동
AND       M00900	// W200 Seleted
AND       M0000A	// OP2 수동 Mode
SET       M00901	// W200 수동 Mode
TON       T0901 1	// W200 수동 Mode
; L8
LOAD NOT  M00008	// OP2 운전준비
OR        T0902	// W200 자동 Mode
RST       M00901	// W200 수동 Mode
; L10
LOAD      M00008	// OP2 운전준비
AND       M00009	// OP2 자동 Mode
AND       M00900	// W200 Seleted
SET       M00902	// W200 자동 Mode
TON       T0902 1	// W200 자동 Mode
; L12
LOAD NOT  M00008	// OP2 운전준비
OR        T0901	// W200 수동 Mode
RST       M00902	// W200 자동 Mode
; L14
LOAD      M00008	// OP2 운전준비
LOAD      M00900	// W200 Seleted
AND       M00902	// W200 자동 Mode
AND       M00908	// W200 정상
AND       P03023	// OP2 자동기동
OR        M00903	// W200 자동기동
AND LOAD
AND NOT   M00904	// W200 자동정지
OUT       M00903	// W200 자동기동
; L16
LOAD NOT  M00910	// W200 비상정지
AND NOT   M00911	// W200 공압이상
AND NOT   M00912	// W200 상부 안전센서 이상
AND NOT   M00913	// W200 하부 안전센서 이상
AND NOT   M00914	// W200 파트이상
AND NOT   M00915	// W200 차종선택 이상
AND NOT   M00916	// W200 이상
AND NOT   M00917	// W200 서보이상
AND NOT   M00918	// W200 서보 근접센서 위치이상
AND NOT   M00919	// W200 서보회전중 L/C 이상
AND NOT   M0091A	// W200 용접로봇 이상
AND NOT   M0091B	// W200 핸드링 로봇 이상
AND NOT   M0091C	// W200 유니트 센서이상
AND NOT   M0091D	// W200 파트센서 체크 이상
AND NOT   M0091E	// W200 슬라이드 안착이상
AND NOT   M0091F	// W200 로보트 인터록 이상
AND NOT   M0099E	// Arc_05 용접누락 이상
AND NOT   M0099F	// Arc_06 용접누락 이상
AND NOT   M00050	// 라인 도어열림
LOAD NOT  M0009B	// 로보트 팬던트 조작 중 장비 정지
OR NOT    M00943	// W200 Work Robot 간섭무
AND LOAD
NOT
LOAD      M00900	// W200 Seleted
AND       M0000A	// OP2 수동 Mode
OR LOAD
OUT       M00904	// W200 자동정지

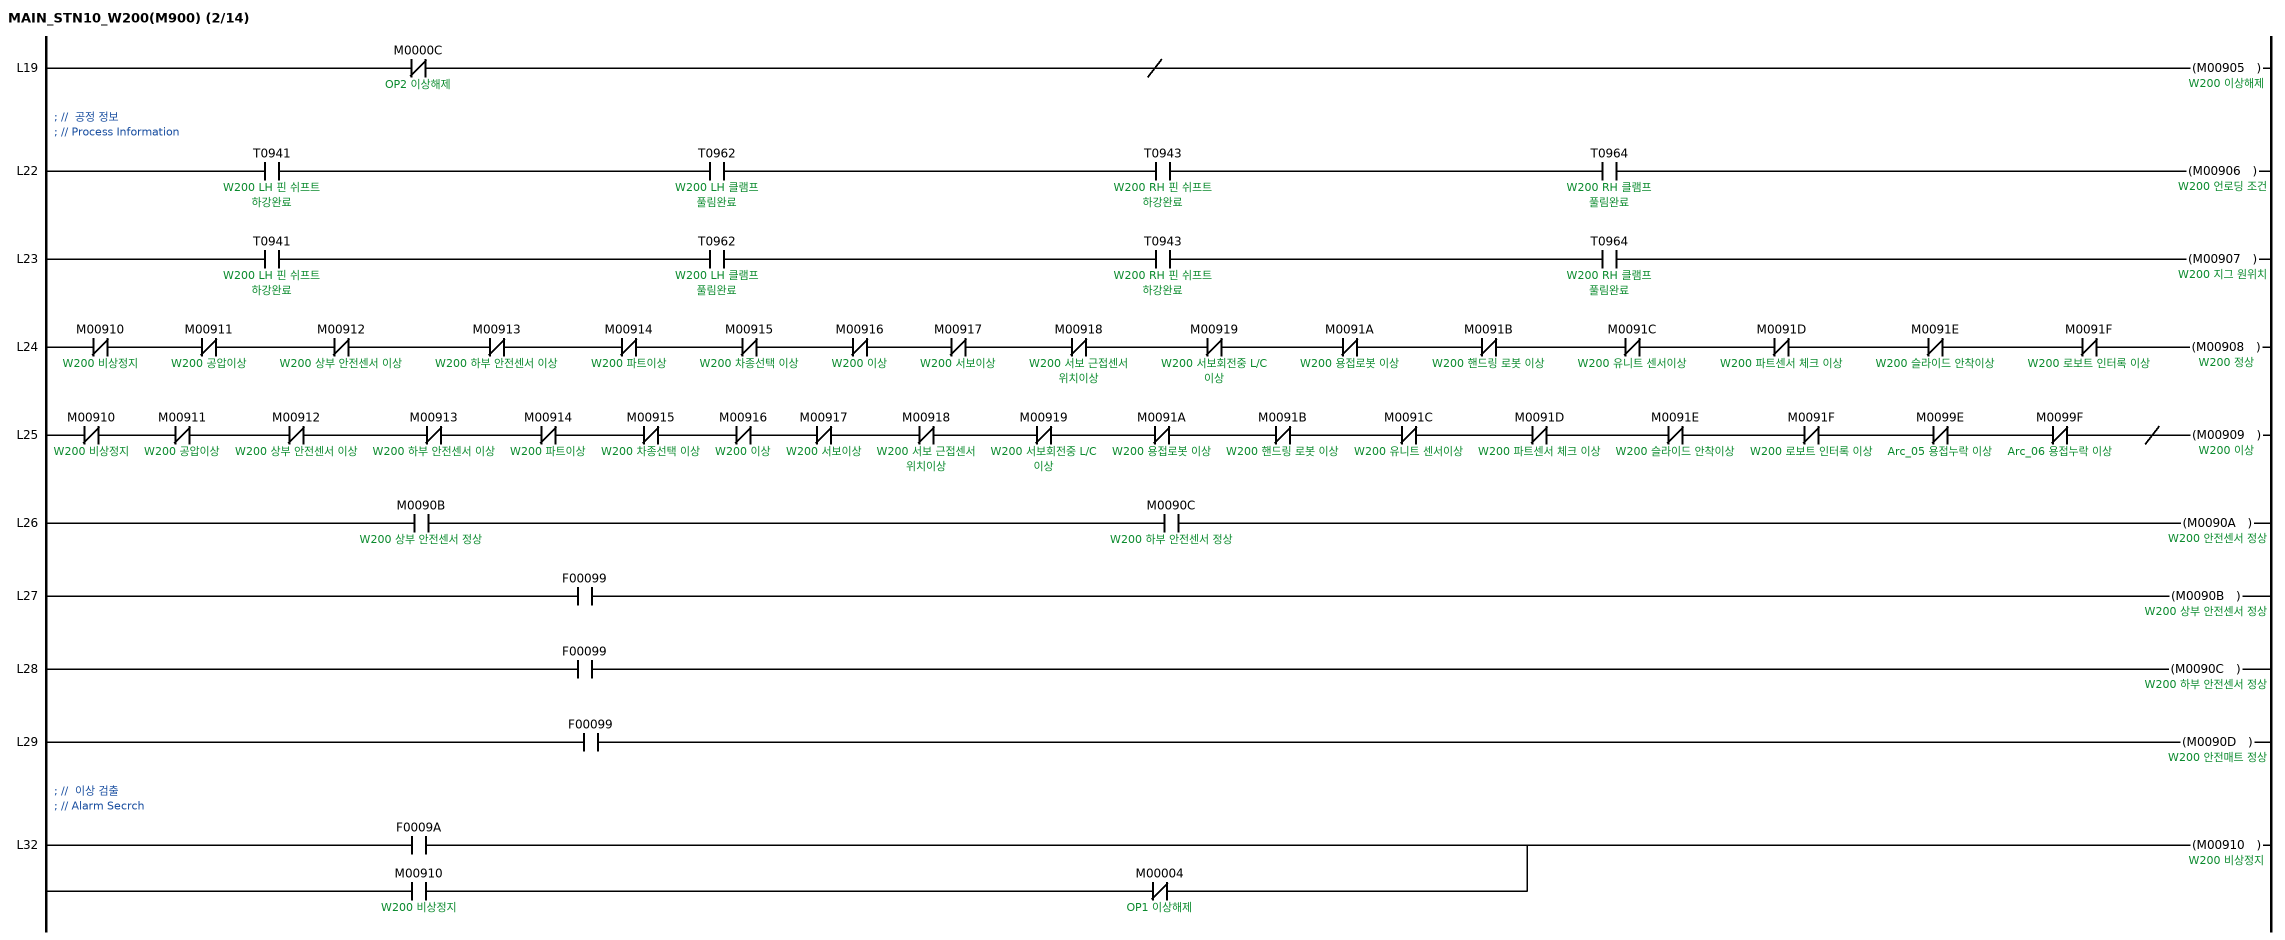
; L19
LOAD NOT  M0000C	// OP2 이상해제
NOT
OUT       M00905	// W200 이상해제
//   //  공정 정보
//   // Process Information
; L22
LOAD      T0941	// W200 LH 핀 쉬프트 하강완료
AND       T0962	// W200 LH 클램프 풀림완료
AND       T0943	// W200 RH 핀 쉬프트 하강완료
AND       T0964	// W200 RH 클램프 풀림완료
OUT       M00906	// W200 언로딩 조건
; L23
LOAD      T0941	// W200 LH 핀 쉬프트 하강완료
AND       T0962	// W200 LH 클램프 풀림완료
AND       T0943	// W200 RH 핀 쉬프트 하강완료
AND       T0964	// W200 RH 클램프 풀림완료
OUT       M00907	// W200 지그 원위치
; L24
LOAD NOT  M00910	// W200 비상정지
AND NOT   M00911	// W200 공압이상
AND NOT   M00912	// W200 상부 안전센서 이상
AND NOT   M00913	// W200 하부 안전센서 이상
AND NOT   M00914	// W200 파트이상
AND NOT   M00915	// W200 차종선택 이상
AND NOT   M00916	// W200 이상
AND NOT   M00917	// W200 서보이상
AND NOT   M00918	// W200 서보 근접센서 위치이상
AND NOT   M00919	// W200 서보회전중 L/C 이상
AND NOT   M0091A	// W200 용접로봇 이상
AND NOT   M0091B	// W200 핸드링 로봇 이상
AND NOT   M0091C	// W200 유니트 센서이상
AND NOT   M0091D	// W200 파트센서 체크 이상
AND NOT   M0091E	// W200 슬라이드 안착이상
AND NOT   M0091F	// W200 로보트 인터록 이상
OUT       M00908	// W200 정상
; L25
LOAD NOT  M00910	// W200 비상정지
AND NOT   M00911	// W200 공압이상
AND NOT   M00912	// W200 상부 안전센서 이상
AND NOT   M00913	// W200 하부 안전센서 이상
AND NOT   M00914	// W200 파트이상
AND NOT   M00915	// W200 차종선택 이상
AND NOT   M00916	// W200 이상
AND NOT   M00917	// W200 서보이상
AND NOT   M00918	// W200 서보 근접센서 위치이상
AND NOT   M00919	// W200 서보회전중 L/C 이상
AND NOT   M0091A	// W200 용접로봇 이상
AND NOT   M0091B	// W200 핸드링 로봇 이상
AND NOT   M0091C	// W200 유니트 센서이상
AND NOT   M0091D	// W200 파트센서 체크 이상
AND NOT   M0091E	// W200 슬라이드 안착이상
AND NOT   M0091F	// W200 로보트 인터록 이상
AND NOT   M0099E	// Arc_05 용접누락 이상
AND NOT   M0099F	// Arc_06 용접누락 이상
NOT
OUT       M00909	// W200 이상
; L26
LOAD      M0090B	// W200 상부 안전센서 정상
AND       M0090C	// W200 하부 안전센서 정상
OUT       M0090A	// W200 안전센서 정상
; L27
LOAD      F00099
OUT       M0090B	// W200 상부 안전센서 정상
; L28
LOAD      F00099
OUT       M0090C	// W200 하부 안전센서 정상
; L29
LOAD      F00099
OUT       M0090D	// W200 안전매트 정상
//   //  이상 검출
//   // Alarm Secrch
; L32
LOAD      F0009A
LOAD      M00910	// W200 비상정지
AND NOT   M00004	// OP1 이상해제
OR LOAD
OUT       M00910	// W200 비상정지

